// TIA Portal V19 export
FUNCTION_BLOCK "FinalCut_FB"   // FB111, LAD
TITLE = GENERIC OLEODINAMIC HEAD MANAGER
// stored: MemoryReserve 100, SetENOAutomatically false
   VAR_INPUT
      AreaInterface : "AreaInterface";
      ZSI : "udt_ZoneSafetyInterface";
      DSI : "udt_DeviceSafetyInterface";
      DataIn : Struct
         CutHead : "ValveMachine_DataIn";
         DrawHead : "ValveMachine_DataIn";
         MarkHead : "ValveMachine_DataIn";
         Locking : "ValveMachine_DataIn";
         Locking_PressureAI : Int;
      END_STRUCT;
      CIn : Struct
         PressureRunning : Bool := FALSE;
         MaterialStandstill : Bool := FALSE;   // FALSE = Either the movement has already started or is about to start
         EnableCutHead : Bool;
         EnableDrawHead : Bool;
         EnableMarkHead : Bool;
         PPrf_PrgNo : DInt;
         CutHead_Manager : "ValveMachine_Manager";
         DrawHead_Manager : "ValveMachine_Manager";
         MarkHead_Manager : "ValveMachine_Manager";
      END_STRUCT;
      Config : Struct
         CheckRestPosition : Bool := TRUE;
         CutHead : "ValveMachine_Config";
         DrawHead : "ValveMachine_Config";
         MarkHead : "ValveMachine_Config";
         Locking : "ValveMachine_Config";
         Locking_AI_HighLimit : Real;
         Locking_AI_LowLimit : Real;
      END_STRUCT;
   END_VAR
   VAR_OUTPUT
      MachineInterface : "MachineInterface";
      DataOut : Struct
         CutHead : "ValveMachine_DataOut";
         DrawHead : "ValveMachine_DataOut";
         MarkHead : "ValveMachine_DataOut";
         Locking : "ValveMachine_DataOut";
      END_STRUCT;
      COut : Struct
         CutHead : "ValveMachine_COut";
         DrawHead : "ValveMachine_COut";
         MarkHead : "ValveMachine_COut";
         Locking : "ValveMachine_COut";
         Avg_R_to_W_Time : Time;
         Avg_W_to_R_Time : Time;
         AllAtRest : Bool;
      END_STRUCT;
   END_VAR
   VAR_IN_OUT
      PersistentValues : "udt_FinalCut_Pers";
   END_VAR
   VAR
      Sts : Struct
         CycleTime : Struct
            CutHead : Struct
               DT_W_Start : DTL;
               DT_W_Stop : DTL;
               DT_R_Start : DTL;
               DT_R_Stop : DTL;
               R_To_W_Exe : Bool;
               W_To_R_Exe : Bool;
               R_To_W_Items : Int;
               R_To_W_Sum : Time;
               W_To_R_Items : Int;
               W_To_R_Sum : Time;
            END_STRUCT;
            DrawHead : Struct
               DT_W_Start : DTL;
               DT_W_Stop : DTL;
               DT_R_Start : DTL;
               DT_R_Stop : DTL;
               R_To_W_Exe : Bool;
               W_To_R_Exe : Bool;
               R_To_W_Items : Int;
               R_To_W_Sum : Time;
               W_To_R_Items : Int;
               W_To_R_Sum : Time;
            END_STRUCT;
            MarkHead : Struct
               DT_W_Start : DTL;
               DT_W_Stop : DTL;
               DT_R_Start : DTL;
               DT_R_Stop : DTL;
               R_To_W_Exe : Bool;
               W_To_R_Exe : Bool;
               R_To_W_Items : Int;
               R_To_W_Sum : Time;
               W_To_R_Items : Int;
               W_To_R_Sum : Time;
            END_STRUCT;
            PPrf_PrgNoSave : DInt;
         END_STRUCT;
         LockingPressure : Real;
         WorkPressureOk : Bool;
         MinPressureOk : Bool;
      END_STRUCT;
      Ctrl : Struct
         Reload : Struct
            CutHead : Bool;
            DrawHead : Bool;
            MarkHead : Bool;
            Locking : Bool;
         END_STRUCT;
         RstAlarms : Bool;
      END_STRUCT;
      Alarm : Struct
         CutHead : "ValveAlr";
         DrawHead : "ValveAlr";
         MarkHead : "ValveAlr";
         Locking : "ValveAlr";
         Locking_NotAWork : Bool;
      END_STRUCT;
      Warning : Struct
         CutHead : "ValveMachine_Wng";
         DrawHead : "ValveMachine_Wng";
         MarkHead : "ValveMachine_Wng";
         Locking : "ValveMachine_Wng";
         CutHead_NotAtRest : Bool := FALSE;
         DrawHead_NotAtRest : Bool;
         MarkHead_NotAtRest : Bool;
         Locking_NotAWork : Bool;
         MaterialNotStandstill : Bool := FALSE;
      END_STRUCT;
      HMI : Struct
         CutHead : Struct
            Last_R_to_W_ID : DInt;
            Last_R_to_W_Time : Time;
            Last_W_to_R_ID : DInt;
            Last_W_to_R_Time : Time;
            Avg_R_to_W_Time : Time;
            Avg_W_to_R_Time : Time;
            Buffer_R_to_W_Time : Array[1..#BUFFER_ITEMS] of Struct
               ID : DInt;
               Value : Time;
            END_STRUCT;
            Buffer_W_to_R_Time : Array[1..#BUFFER_ITEMS] of Struct
               ID : DInt;
               Value : Time;
            END_STRUCT;
         END_STRUCT;
         DrawHead : Struct
            Last_R_to_W_ID : DInt;
            Last_R_to_W_Time : Time;
            Last_W_to_R_ID : DInt;
            Last_W_to_R_Time : Time;
            Avg_R_to_W_Time : Time;
            Avg_W_to_R_Time : Time;
            Buffer_R_to_W_Time : Array[1..#BUFFER_ITEMS] of Struct
               ID : DInt;
               Value : Time;
            END_STRUCT;
            Buffer_W_to_R_Time : Array[1..#BUFFER_ITEMS] of Struct
               ID : DInt;
               Value : Time;
            END_STRUCT;
         END_STRUCT;
         MarkHead : Struct
            Last_R_to_W_ID : DInt;
            Last_R_to_W_Time : Time;
            Last_W_to_R_ID : DInt;
            Last_W_to_R_Time : Time;
            Avg_R_to_W_Time : Time;
            Avg_W_to_R_Time : Time;
            Buffer_R_to_W_Time : Array[1..#BUFFER_ITEMS] of Struct
               ID : DInt;
               Value : Time;
            END_STRUCT;
            Buffer_W_to_R_Time : Array[1..#BUFFER_ITEMS] of Struct
               ID : DInt;
               Value : Time;
            END_STRUCT;
         END_STRUCT;
      END_STRUCT;
      CutHead : "ValveMachine_FB";
      DrawHead : "ValveMachine_FB";
      MarkHead : "ValveMachine_FB";
      Locking : "ValveMachine_FB";
      TON_CutHead_Pause : IEC_TIMER;
      TON_CutHead_Duration : IEC_TIMER;
      TON_DrawHead_Pause : IEC_TIMER;
      TON_DrawHead_Duration : IEC_TIMER;
      TON_MarkHead_Pause : IEC_TIMER;
      TON_MarkHead_Duration : IEC_TIMER;
      TON_LockingTimeOut : IEC_TIMER;
      PE_Aux : Struct
         CutHead : Struct
            AtRest : Bool;
            AtWork : Bool;
            NotAtRest : Bool;
            NotAtWork : Bool;
         END_STRUCT;
         DrawHead : Struct
            AtRest : Bool;
            AtWork : Bool;
            NotAtRest : Bool;
            NotAtWork : Bool;
         END_STRUCT;
         MarkHead : Struct
            AtRest : Bool;
            AtWork : Bool;
            NotAtRest : Bool;
            NotAtWork : Bool;
         END_STRUCT;
      END_STRUCT;
      i : Int;
   END_VAR
   VAR_TEMP
      PE : Struct
         CutHead : Struct
            AtRest : Bool;
            AtWork : Bool;
            NotAtRest : Bool;
            NotAtWork : Bool;
         END_STRUCT;
         DrawHead : Struct
            AtRest : Bool;
            AtWork : Bool;
            NotAtRest : Bool;
            NotAtWork : Bool;
         END_STRUCT;
         MarkHead : Struct
            AtRest : Bool;
            AtWork : Bool;
            NotAtRest : Bool;
            NotAtWork : Bool;
         END_STRUCT;
      END_STRUCT;
      ReturnVal : Word;
      ScaleRetVal : Word;
   END_VAR
   VAR CONSTANT
      BUFFER_ITEMS : Int := 10;
   END_VAR
   VAR_TEMP   // added for the SCL form of the ladder/FBD networks
      _w1 : Bool;
      _w2 : Bool;
      _w3 : Bool;
      _w4 : Bool;
   END_VAR
BEGIN

REGION Network 1 (SCL): Reset alarms
   #Ctrl.RstAlarms := #AreaInterface.RstAlarms;

   IF    #Ctrl.RstAlarms THEN

       #Alarm.Locking_NotAWork := FALSE;

   END_IF;
END_REGION

REGION Network 2: >
END_REGION

REGION Network 3: <<< CUT HEAD >>>
END_REGION

REGION Network 4: Pressure reload for avoiding losing of rest position cause leakage on hydraulic cylinders
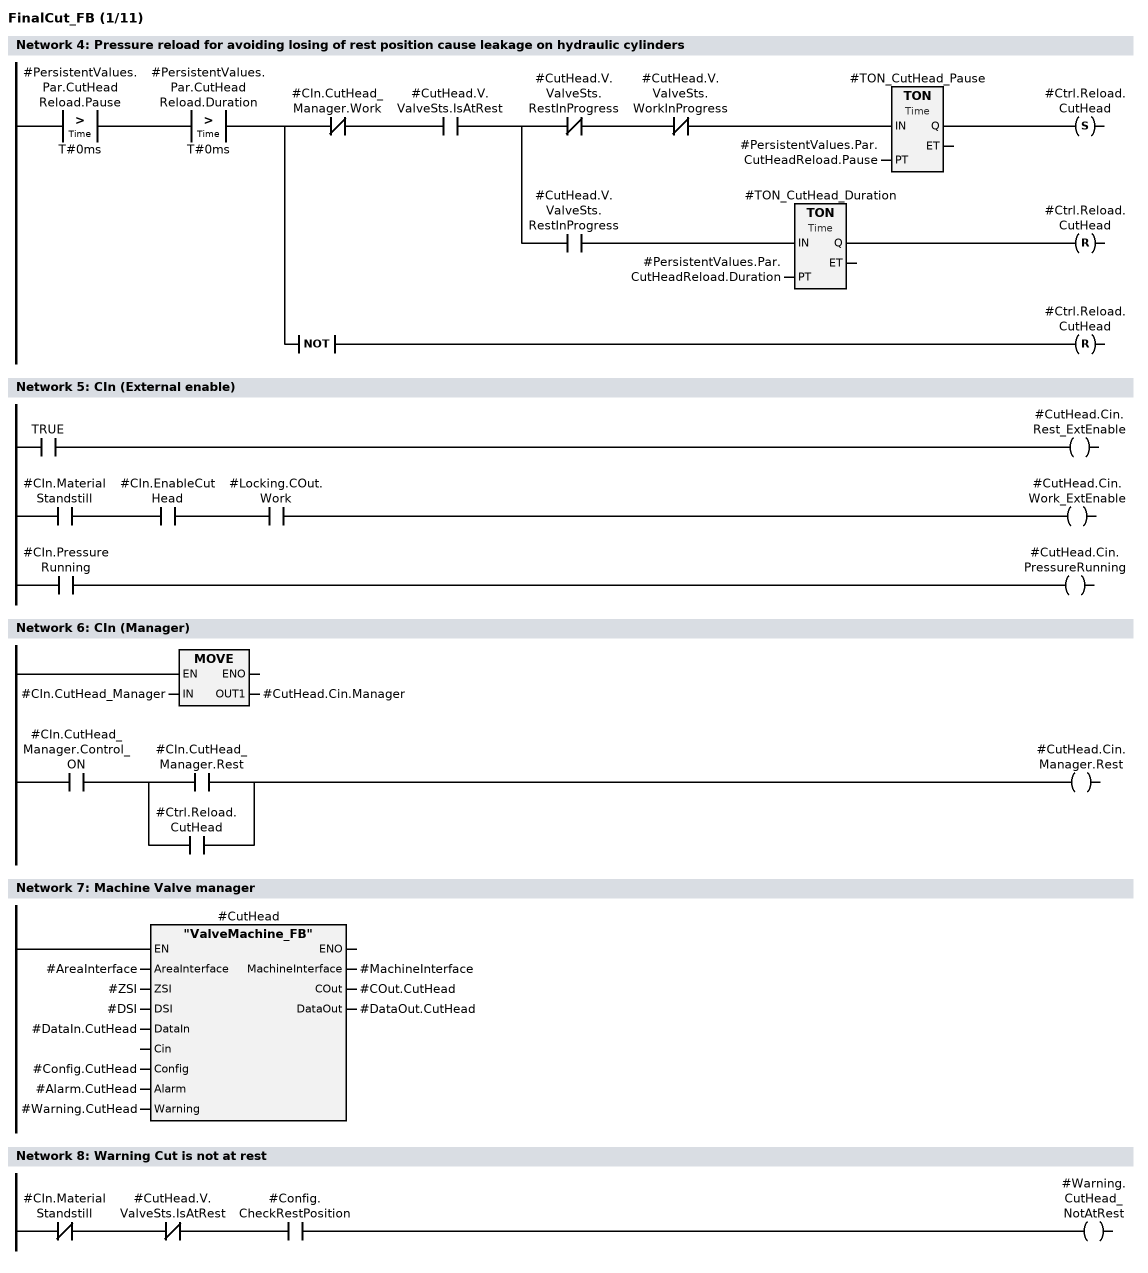
   RUNG wire#powerrail
      { S7_Templates := "SrcType := Time" } GT_Contact(in1 := #PersistentValues.Par.CutHeadReload.Pause, in2 := T#0ms)
      { S7_Templates := "SrcType := Time" } GT_Contact(in1 := #PersistentValues.Par.CutHeadReload.Duration, in2 := T#0ms)
      wire#w1
      I_Contact( #CIn.CutHead_Manager.Work )
      Contact( #CutHead.V.ValveSts.IsAtRest )
      wire#w2
      I_Contact( #CutHead.V.ValveSts.RestInProgress )
      I_Contact( #CutHead.V.ValveSts.WorkInProgress )
      { S7_Templates := "time_type := Time" } #TON_CutHead_Pause.TON(pt := #PersistentValues.Par.CutHeadReload.Pause, et =>)
      S_Coil( #Ctrl.Reload.CutHead )
   END_RUNG
   RUNG wire#w2
      Contact( #CutHead.V.ValveSts.RestInProgress )
      { S7_Templates := "time_type := Time" } #TON_CutHead_Duration.TON(pt := #PersistentValues.Par.CutHeadReload.Duration, et =>)
      R_Coil( #Ctrl.Reload.CutHead )
   END_RUNG
   RUNG wire#w1
      Not()
      R_Coil( #Ctrl.Reload.CutHead )
   END_RUNG
   // the same network as SCL:
   #_w1 := (#PersistentValues.Par.CutHeadReload.Pause > T#0ms) AND (#PersistentValues.Par.CutHeadReload.Duration > T#0ms);
   #_w2 := #_w1 AND NOT #CIn.CutHead_Manager.Work AND #CutHead.V.ValveSts.IsAtRest;
   #TON_CutHead_Pause.TON(IN := #_w2 AND NOT #CutHead.V.ValveSts.RestInProgress AND NOT #CutHead.V.ValveSts.WorkInProgress,
                          PT := #PersistentValues.Par.CutHeadReload.Pause);
   IF #TON_CutHead_Pause.Q THEN #Ctrl.Reload.CutHead := TRUE; END_IF;
   #TON_CutHead_Duration.TON(IN := #_w2 AND #CutHead.V.ValveSts.RestInProgress,
                           PT := #PersistentValues.Par.CutHeadReload.Duration);
   IF #TON_CutHead_Duration.Q THEN #Ctrl.Reload.CutHead := FALSE; END_IF;
   IF NOT #_w1 THEN #Ctrl.Reload.CutHead := FALSE; END_IF;
END_REGION

REGION Network 5: CIn (External enable)
   RUNG wire#powerrail
      Contact( TRUE )
      Coil( #CutHead.Cin.Rest_ExtEnable )
   END_RUNG
   RUNG wire#powerrail
      Contact( #CIn.MaterialStandstill )
      Contact( #CIn.EnableCutHead )
      Contact( #Locking.COut.Work )
      Coil( #CutHead.Cin.Work_ExtEnable )
   END_RUNG
   RUNG wire#powerrail
      Contact( #CIn.PressureRunning )
      Coil( #CutHead.Cin.PressureRunning )
   END_RUNG
   // the same network as SCL:
   #CutHead.Cin.Rest_ExtEnable := TRUE;
   #CutHead.Cin.Work_ExtEnable := #CIn.MaterialStandstill AND #CIn.EnableCutHead AND #Locking.COut.Work;
   #CutHead.Cin.PressureRunning := #CIn.PressureRunning;
END_REGION

REGION Network 6: CIn (Manager)
   RUNG wire#powerrail
      Move(in := #CIn.CutHead_Manager, out1 => #CutHead.Cin.Manager)
   END_RUNG
   RUNG wire#powerrail
      Contact( #CIn.CutHead_Manager.Control_ON )
      wire#w1
      Contact( #CIn.CutHead_Manager.Rest )
      wire#w2
      Coil( #CutHead.Cin.Manager.Rest )
   END_RUNG
   RUNG wire#w1
      Contact( #Ctrl.Reload.CutHead )
   END_RUNG wire#w2
   // the same network as SCL:
   #CutHead.Cin.Manager := #CIn.CutHead_Manager;
   #CutHead.Cin.Manager.Rest := #CIn.CutHead_Manager.Control_ON AND (#CIn.CutHead_Manager.Rest OR #Ctrl.Reload.CutHead);
END_REGION

REGION Network 7: Machine Valve manager
   RUNG wire#powerrail
      #CutHead(AreaInterface := #AreaInterface, ZSI := #ZSI, DSI := #DSI, DataIn := #DataIn.CutHead, Cin :=, Config := #Config.CutHead, Alarm := #Alarm.CutHead, Warning := #Warning.CutHead, MachineInterface => #MachineInterface, COut => #COut.CutHead, DataOut => #DataOut.CutHead)
   END_RUNG
   // the same network as SCL:
   #CutHead(AreaInterface := #AreaInterface,   // "ValveMachine_FB"
            ZSI := #ZSI,
            DSI := #DSI,
            DataIn := #DataIn.CutHead,
            Config := #Config.CutHead,
            Alarm := #Alarm.CutHead,
            Warning := #Warning.CutHead,
            MachineInterface => #MachineInterface,
            COut => #COut.CutHead,
            DataOut => #DataOut.CutHead);
END_REGION

REGION Network 8: Warning Cut is not at rest
   RUNG wire#powerrail
      I_Contact( #CIn.MaterialStandstill )
      I_Contact( #CutHead.V.ValveSts.IsAtRest )
      Contact( #Config.CheckRestPosition )
      Coil( #Warning.CutHead_NotAtRest )
   END_RUNG
   // the same network as SCL:
   #Warning.CutHead_NotAtRest := NOT #CIn.MaterialStandstill AND NOT #CutHead.V.ValveSts.IsAtRest AND #Config.CheckRestPosition;
END_REGION

REGION Network 9: At Rest / At work positive/negative edge
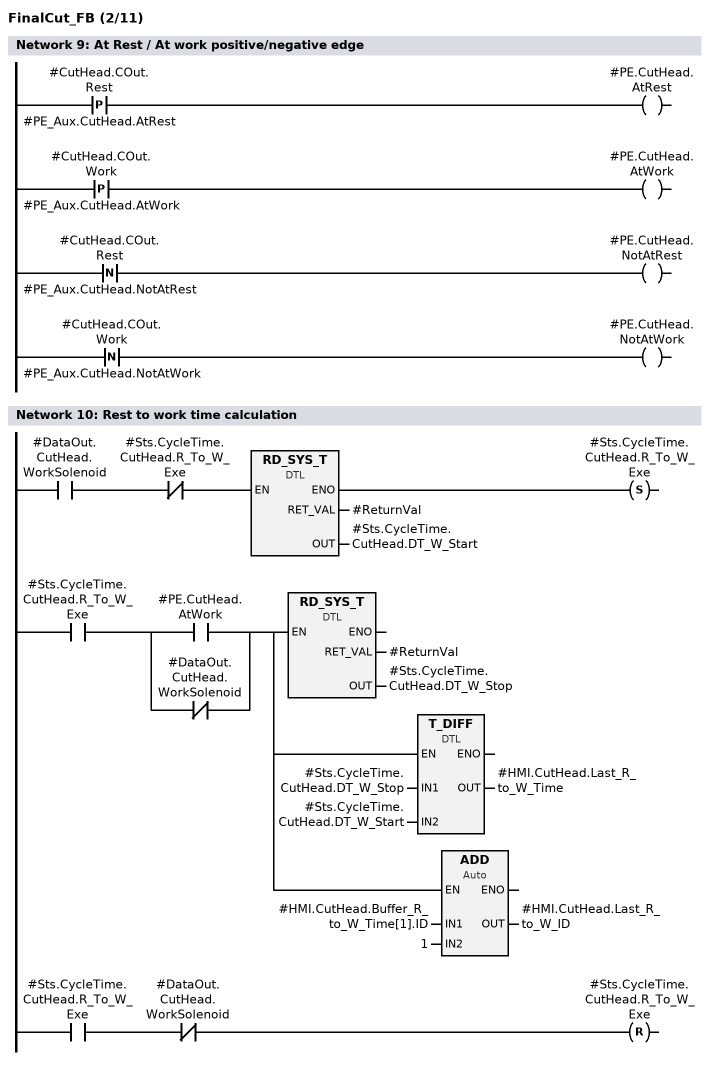
   RUNG wire#powerrail
      P_Contact(operand := #CutHead.COut.Rest, bit := #PE_Aux.CutHead.AtRest)
      Coil( #PE.CutHead.AtRest )
   END_RUNG
   RUNG wire#powerrail
      P_Contact(operand := #CutHead.COut.Work, bit := #PE_Aux.CutHead.AtWork)
      Coil( #PE.CutHead.AtWork )
   END_RUNG
   RUNG wire#powerrail
      N_Contact(operand := #CutHead.COut.Rest, bit := #PE_Aux.CutHead.NotAtRest)
      Coil( #PE.CutHead.NotAtRest )
   END_RUNG
   RUNG wire#powerrail
      N_Contact(operand := #CutHead.COut.Work, bit := #PE_Aux.CutHead.NotAtWork)
      Coil( #PE.CutHead.NotAtWork )
   END_RUNG
   // the same network as SCL:
   #_w1 := #CutHead.COut.Rest AND NOT #PE_Aux.CutHead.AtRest;   // rising edge of #CutHead.COut.Rest
   #PE_Aux.CutHead.AtRest := #CutHead.COut.Rest;
   #PE.CutHead.AtRest := #_w1;
   #_w2 := #CutHead.COut.Work AND NOT #PE_Aux.CutHead.AtWork;   // rising edge of #CutHead.COut.Work
   #PE_Aux.CutHead.AtWork := #CutHead.COut.Work;
   #PE.CutHead.AtWork := #_w2;
   #_w3 := NOT #CutHead.COut.Rest AND #PE_Aux.CutHead.NotAtRest;   // falling edge of #CutHead.COut.Rest
   #PE_Aux.CutHead.NotAtRest := #CutHead.COut.Rest;
   #PE.CutHead.NotAtRest := #_w3;
   #_w4 := NOT #CutHead.COut.Work AND #PE_Aux.CutHead.NotAtWork;   // falling edge of #CutHead.COut.Work
   #PE_Aux.CutHead.NotAtWork := #CutHead.COut.Work;
   #PE.CutHead.NotAtWork := #_w4;
END_REGION

REGION Network 10: Rest to work time calculation
   RUNG wire#powerrail
      Contact( #DataOut.CutHead.WorkSolenoid )
      I_Contact( #Sts.CycleTime.CutHead.R_To_W_Exe )
      { S7_Templates := "date_type := DTL" } RD_SYS_T(RET_VAL => #ReturnVal, OUT => #Sts.CycleTime.CutHead.DT_W_Start)
      S_Coil( #Sts.CycleTime.CutHead.R_To_W_Exe )
   END_RUNG
   RUNG wire#powerrail
      Contact( #Sts.CycleTime.CutHead.R_To_W_Exe )
      wire#w1
      Contact( #PE.CutHead.AtWork )
      wire#w2
      { S7_Templates := "date_type := DTL" } RD_SYS_T(RET_VAL => #ReturnVal, OUT => #Sts.CycleTime.CutHead.DT_W_Stop)
   END_RUNG
   RUNG wire#w1
      I_Contact( #DataOut.CutHead.WorkSolenoid )
   END_RUNG wire#w2
   RUNG wire#w2
      { S7_Templates := "[date_type := DTL, time_type := Time]" } T_DIFF(IN1 := #Sts.CycleTime.CutHead.DT_W_Stop, IN2 := #Sts.CycleTime.CutHead.DT_W_Start, OUT => #HMI.CutHead.Last_R_to_W_Time)
   END_RUNG
   RUNG wire#w2
      Add(in1 := #HMI.CutHead.Buffer_R_to_W_Time[1].ID, in2 := 1, out => #HMI.CutHead.Last_R_to_W_ID)
   END_RUNG
   RUNG wire#powerrail
      Contact( #Sts.CycleTime.CutHead.R_To_W_Exe )
      I_Contact( #DataOut.CutHead.WorkSolenoid )
      R_Coil( #Sts.CycleTime.CutHead.R_To_W_Exe )
   END_RUNG
   // the same network as SCL:
   #ReturnVal := RD_SYS_T(EN := #DataOut.CutHead.WorkSolenoid AND NOT #Sts.CycleTime.CutHead.R_To_W_Exe,
                          OUT => #Sts.CycleTime.CutHead.DT_W_Start,
                          ENO => #_w1);
   IF #_w1 THEN #Sts.CycleTime.CutHead.R_To_W_Exe := TRUE; END_IF;
   IF #Sts.CycleTime.CutHead.R_To_W_Exe AND (#PE.CutHead.AtWork OR NOT #DataOut.CutHead.WorkSolenoid) THEN
       #ReturnVal := RD_SYS_T(OUT => #Sts.CycleTime.CutHead.DT_W_Stop);
       T_DIFF(IN1 := #Sts.CycleTime.CutHead.DT_W_Stop,
              IN2 := #Sts.CycleTime.CutHead.DT_W_Start,
              OUT => #HMI.CutHead.Last_R_to_W_Time);
       #HMI.CutHead.Last_R_to_W_ID := #HMI.CutHead.Buffer_R_to_W_Time[1].ID + 1;
   END_IF;
   IF #Sts.CycleTime.CutHead.R_To_W_Exe AND NOT #DataOut.CutHead.WorkSolenoid THEN
       #Sts.CycleTime.CutHead.R_To_W_Exe := FALSE;
   END_IF;
END_REGION

REGION Network 11: Work to rest time calculation
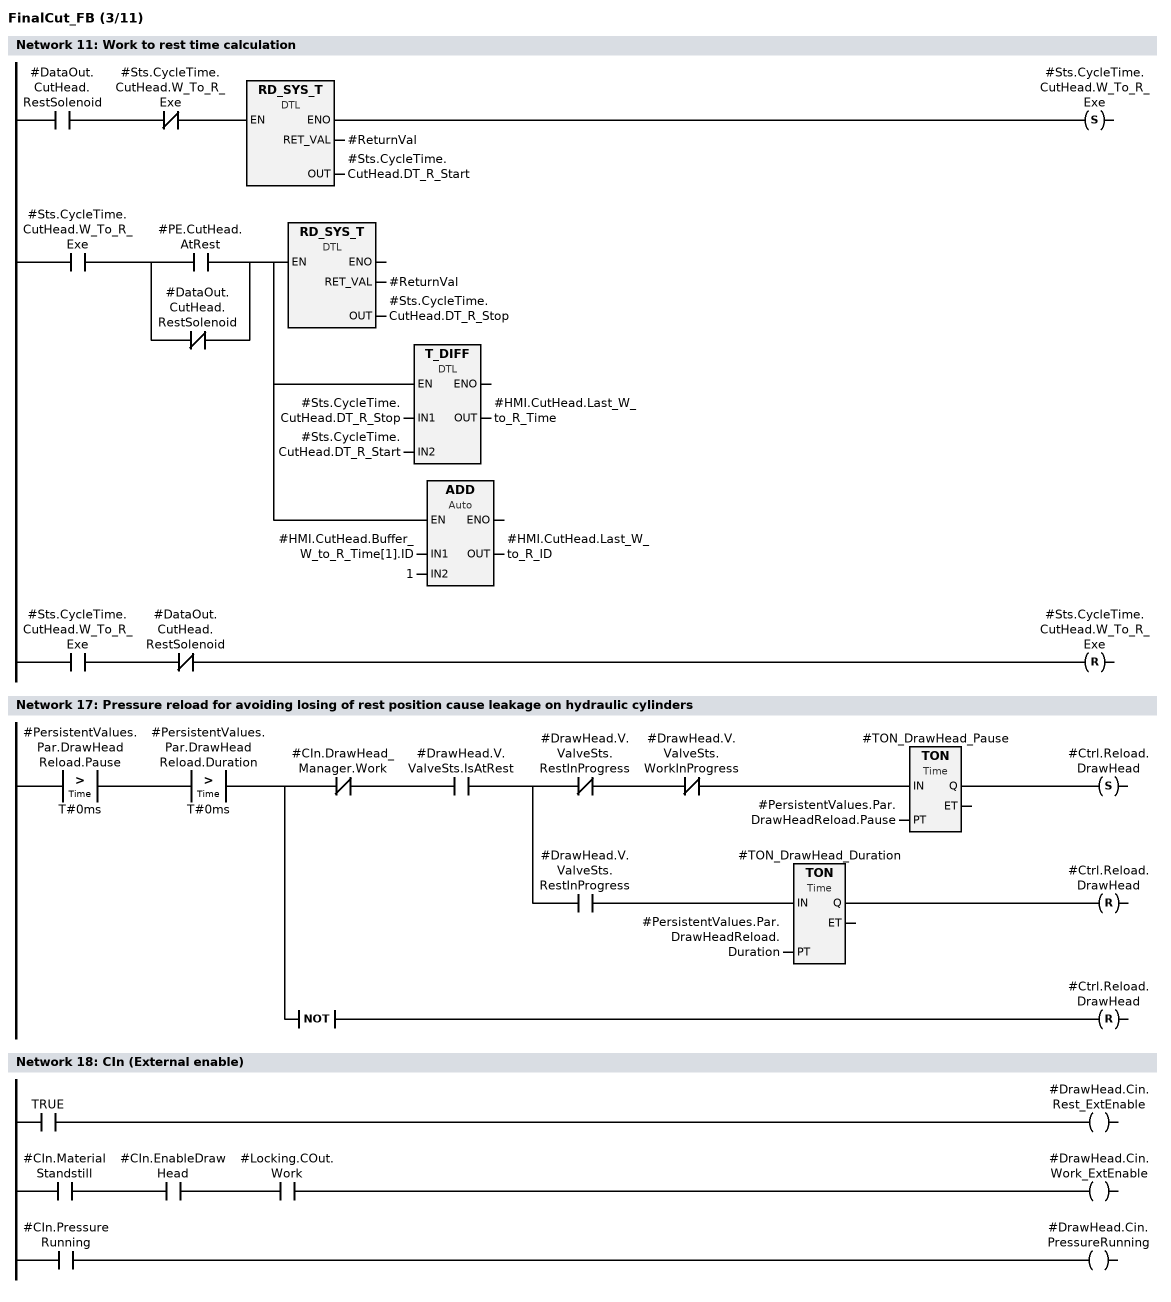
   RUNG wire#powerrail
      Contact( #DataOut.CutHead.RestSolenoid )
      I_Contact( #Sts.CycleTime.CutHead.W_To_R_Exe )
      { S7_Templates := "date_type := DTL" } RD_SYS_T(RET_VAL => #ReturnVal, OUT => #Sts.CycleTime.CutHead.DT_R_Start)
      S_Coil( #Sts.CycleTime.CutHead.W_To_R_Exe )
   END_RUNG
   RUNG wire#powerrail
      Contact( #Sts.CycleTime.CutHead.W_To_R_Exe )
      wire#w1
      Contact( #PE.CutHead.AtRest )
      wire#w2
      { S7_Templates := "date_type := DTL" } RD_SYS_T(RET_VAL => #ReturnVal, OUT => #Sts.CycleTime.CutHead.DT_R_Stop)
   END_RUNG
   RUNG wire#w1
      I_Contact( #DataOut.CutHead.RestSolenoid )
   END_RUNG wire#w2
   RUNG wire#w2
      { S7_Templates := "[date_type := DTL, time_type := Time]" } T_DIFF(IN1 := #Sts.CycleTime.CutHead.DT_R_Stop, IN2 := #Sts.CycleTime.CutHead.DT_R_Start, OUT => #HMI.CutHead.Last_W_to_R_Time)
   END_RUNG
   RUNG wire#w2
      Add(in1 := #HMI.CutHead.Buffer_W_to_R_Time[1].ID, in2 := 1, out => #HMI.CutHead.Last_W_to_R_ID)
   END_RUNG
   RUNG wire#powerrail
      Contact( #Sts.CycleTime.CutHead.W_To_R_Exe )
      I_Contact( #DataOut.CutHead.RestSolenoid )
      R_Coil( #Sts.CycleTime.CutHead.W_To_R_Exe )
   END_RUNG
   // the same network as SCL:
   #ReturnVal := RD_SYS_T(EN := #DataOut.CutHead.RestSolenoid AND NOT #Sts.CycleTime.CutHead.W_To_R_Exe,
                          OUT => #Sts.CycleTime.CutHead.DT_R_Start,
                          ENO => #_w1);
   IF #_w1 THEN #Sts.CycleTime.CutHead.W_To_R_Exe := TRUE; END_IF;
   IF #Sts.CycleTime.CutHead.W_To_R_Exe AND (#PE.CutHead.AtRest OR NOT #DataOut.CutHead.RestSolenoid) THEN
       #ReturnVal := RD_SYS_T(OUT => #Sts.CycleTime.CutHead.DT_R_Stop);
       T_DIFF(IN1 := #Sts.CycleTime.CutHead.DT_R_Stop,
              IN2 := #Sts.CycleTime.CutHead.DT_R_Start,
              OUT => #HMI.CutHead.Last_W_to_R_Time);
       #HMI.CutHead.Last_W_to_R_ID := #HMI.CutHead.Buffer_W_to_R_Time[1].ID + 1;
   END_IF;
   IF #Sts.CycleTime.CutHead.W_To_R_Exe AND NOT #DataOut.CutHead.RestSolenoid THEN
       #Sts.CycleTime.CutHead.W_To_R_Exe := FALSE;
   END_IF;
END_REGION

REGION Network 12 (SCL): Init buffers & average calculations
   IF #CIn.PPrf_PrgNo <> #Sts.CycleTime.PPrf_PrgNoSave OR #CIn.PPrf_PrgNo <= 0 THEN

       FOR #i := 1 TO #BUFFER_ITEMS DO
           #HMI.CutHead.Buffer_R_to_W_Time[#i].ID := 0;
           #HMI.CutHead.Buffer_R_to_W_Time[#i].Value := T#0s;
           #HMI.CutHead.Buffer_W_to_R_Time[#i].ID := 0;
           #HMI.CutHead.Buffer_W_to_R_Time[#i].Value := T#0s;
       END_FOR;

       #HMI.CutHead.Last_R_to_W_ID := 0;
       #HMI.CutHead.Last_R_to_W_Time := T#0ms;
       #HMI.CutHead.Avg_R_to_W_Time := #Config.CutHead.V.WorkTimeOut;

       #HMI.CutHead.Last_W_to_R_ID := 0;
       #HMI.CutHead.Last_W_to_R_Time := T#0ms;
       #HMI.CutHead.Avg_W_to_R_Time := #Config.CutHead.V.RestTimeOut;

   END_IF;


   #Sts.CycleTime.PPrf_PrgNoSave := #CIn.PPrf_PrgNo;
END_REGION

REGION Network 13 (SCL): Add new items to Rest-TO-Work buffer & calculate average

   IF #HMI.CutHead.Last_R_to_W_Time >= #CutHead.Config.V.WorkTimeOut OR #Alarm.CutHead.TimeOutWork THEN

       #HMI.CutHead.Last_R_to_W_ID := -1; // Force red background on the HMI visualization



   ELSIF #HMI.CutHead.Last_R_to_W_ID <> #HMI.CutHead.Buffer_R_to_W_Time[1].ID AND #HMI.CutHead.Last_R_to_W_Time < #CutHead.Config.V.WorkTimeOut AND #HMI.CutHead.Last_R_to_W_Time > T#0ms THEN

       #i := #BUFFER_ITEMS;

       WHILE #i >= 2 DO

           #HMI.CutHead.Buffer_R_to_W_Time[#i] := #HMI.CutHead.Buffer_R_to_W_Time[#i - 1];

           #i -= 1;

       END_WHILE;

       #HMI.CutHead.Buffer_R_to_W_Time[1].ID := #HMI.CutHead.Last_R_to_W_ID;
       #HMI.CutHead.Buffer_R_to_W_Time[1].Value := #HMI.CutHead.Last_R_to_W_Time;

       #Sts.CycleTime.CutHead.R_To_W_Items := 0;
       #Sts.CycleTime.CutHead.R_To_W_Sum := T#0s;


       FOR #i := 1 TO #BUFFER_ITEMS DO

           IF #HMI.CutHead.Buffer_R_to_W_Time[#i].ID > 0 AND #HMI.CutHead.Buffer_R_to_W_Time[#i].Value > T#0ms THEN
               #Sts.CycleTime.CutHead.R_To_W_Items += 1;
               #Sts.CycleTime.CutHead.R_To_W_Sum := #Sts.CycleTime.CutHead.R_To_W_Sum + #HMI.CutHead.Buffer_R_to_W_Time[#i].Value;
           END_IF;

       END_FOR;

       IF #Sts.CycleTime.CutHead.R_To_W_Items >= 5 THEN
           #HMI.CutHead.Avg_R_to_W_Time := #Sts.CycleTime.CutHead.R_To_W_Sum / #Sts.CycleTime.CutHead.R_To_W_Items;
       ELSE
           #HMI.CutHead.Avg_R_to_W_Time := #Config.CutHead.V.WorkTimeOut;
       END_IF;

   END_IF;
END_REGION

REGION Network 14 (SCL): Add new items to Work-TO-Rest buffer & calculate average
   IF #HMI.CutHead.Last_W_to_R_Time >= #CutHead.Config.V.RestTimeOut OR #Alarm.CutHead.TimeOutRest THEN

       #HMI.CutHead.Last_W_to_R_ID := -1; // Force red background on the HMI visualization

   ELSIF #HMI.CutHead.Last_W_to_R_ID <> #HMI.CutHead.Buffer_W_to_R_Time[1].ID AND #HMI.CutHead.Last_W_to_R_Time < #CutHead.Config.V.RestTimeOut AND #HMI.CutHead.Last_W_to_R_Time > T#0ms  THEN

       #i := #BUFFER_ITEMS;

       WHILE #i >= 2 DO

           #HMI.CutHead.Buffer_W_to_R_Time[#i] := #HMI.CutHead.Buffer_W_to_R_Time[#i - 1];

           #i -= 1;

       END_WHILE;

       #HMI.CutHead.Buffer_W_to_R_Time[1].ID := #HMI.CutHead.Last_W_to_R_ID;
       #HMI.CutHead.Buffer_W_to_R_Time[1].Value := #HMI.CutHead.Last_W_to_R_Time;

       #Sts.CycleTime.CutHead.W_To_R_Items := 0;
       #Sts.CycleTime.CutHead.W_To_R_Sum := T#0s;


       FOR #i := 1 TO #BUFFER_ITEMS DO

           IF #HMI.CutHead.Buffer_W_to_R_Time[#i].ID > 0 AND #HMI.CutHead.Buffer_W_to_R_Time[#i].Value > T#0ms  THEN
               #Sts.CycleTime.CutHead.W_To_R_Items += 1;
               #Sts.CycleTime.CutHead.W_To_R_Sum := #Sts.CycleTime.CutHead.W_To_R_Sum + #HMI.CutHead.Buffer_W_to_R_Time[#i].Value;
           END_IF;

       END_FOR;

       IF #Sts.CycleTime.CutHead.W_To_R_Items >= 5 THEN
           #HMI.CutHead.Avg_W_to_R_Time := #Sts.CycleTime.CutHead.W_To_R_Sum / #Sts.CycleTime.CutHead.W_To_R_Items;
       ELSE
           #HMI.CutHead.Avg_W_to_R_Time := #Config.CutHead.V.RestTimeOut;
       END_IF;

   END_IF;
END_REGION

REGION Network 15: >
END_REGION

REGION Network 16: <<< DRAWING HEAD >>>
END_REGION

REGION Network 17: Pressure reload for avoiding losing of rest position cause leakage on hydraulic cylinders
   RUNG wire#powerrail
      { S7_Templates := "SrcType := Time" } GT_Contact(in1 := #PersistentValues.Par.DrawHeadReload.Pause, in2 := T#0ms)
      { S7_Templates := "SrcType := Time" } GT_Contact(in1 := #PersistentValues.Par.DrawHeadReload.Duration, in2 := T#0ms)
      wire#w1
      I_Contact( #CIn.DrawHead_Manager.Work )
      Contact( #DrawHead.V.ValveSts.IsAtRest )
      wire#w2
      I_Contact( #DrawHead.V.ValveSts.RestInProgress )
      I_Contact( #DrawHead.V.ValveSts.WorkInProgress )
      { S7_Templates := "time_type := Time" } #TON_DrawHead_Pause.TON(pt := #PersistentValues.Par.DrawHeadReload.Pause, et =>)
      S_Coil( #Ctrl.Reload.DrawHead )
   END_RUNG
   RUNG wire#w2
      Contact( #DrawHead.V.ValveSts.RestInProgress )
      { S7_Templates := "time_type := Time" } #TON_DrawHead_Duration.TON(pt := #PersistentValues.Par.DrawHeadReload.Duration, et =>)
      R_Coil( #Ctrl.Reload.DrawHead )
   END_RUNG
   RUNG wire#w1
      Not()
      R_Coil( #Ctrl.Reload.DrawHead )
   END_RUNG
   // the same network as SCL:
   #_w1 := (#PersistentValues.Par.DrawHeadReload.Pause > T#0ms) AND (#PersistentValues.Par.DrawHeadReload.Duration > T#0ms);
   #_w2 := #_w1 AND NOT #CIn.DrawHead_Manager.Work AND #DrawHead.V.ValveSts.IsAtRest;
   #TON_DrawHead_Pause.TON(IN := #_w2 AND NOT #DrawHead.V.ValveSts.RestInProgress AND NOT #DrawHead.V.ValveSts.WorkInProgress,
                           PT := #PersistentValues.Par.DrawHeadReload.Pause);
   IF #TON_DrawHead_Pause.Q THEN #Ctrl.Reload.DrawHead := TRUE; END_IF;
   #TON_DrawHead_Duration.TON(IN := #_w2 AND #DrawHead.V.ValveSts.RestInProgress,
                           PT := #PersistentValues.Par.DrawHeadReload.Duration);
   IF #TON_DrawHead_Duration.Q THEN #Ctrl.Reload.DrawHead := FALSE; END_IF;
   IF NOT #_w1 THEN #Ctrl.Reload.DrawHead := FALSE; END_IF;
END_REGION

REGION Network 18: CIn (External enable)
   RUNG wire#powerrail
      Contact( TRUE )
      Coil( #DrawHead.Cin.Rest_ExtEnable )
   END_RUNG
   RUNG wire#powerrail
      Contact( #CIn.MaterialStandstill )
      Contact( #CIn.EnableDrawHead )
      Contact( #Locking.COut.Work )
      Coil( #DrawHead.Cin.Work_ExtEnable )
   END_RUNG
   RUNG wire#powerrail
      Contact( #CIn.PressureRunning )
      Coil( #DrawHead.Cin.PressureRunning )
   END_RUNG
   // the same network as SCL:
   #DrawHead.Cin.Rest_ExtEnable := TRUE;
   #DrawHead.Cin.Work_ExtEnable := #CIn.MaterialStandstill AND #CIn.EnableDrawHead AND #Locking.COut.Work;
   #DrawHead.Cin.PressureRunning := #CIn.PressureRunning;
END_REGION

REGION Network 19: CIn (Manager)
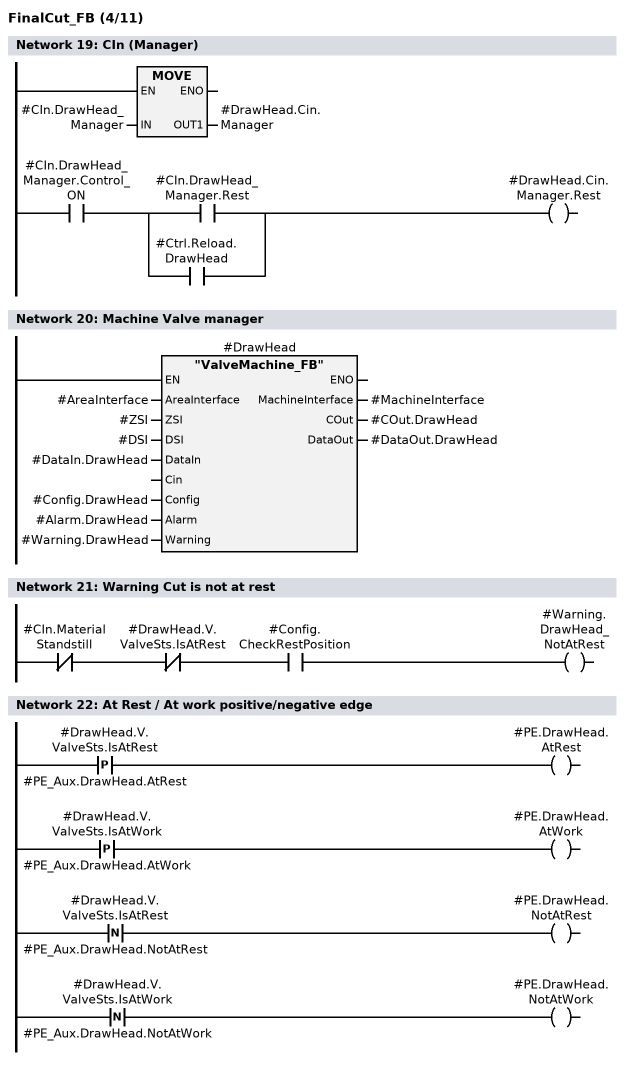
   RUNG wire#powerrail
      Move(in := #CIn.DrawHead_Manager, out1 => #DrawHead.Cin.Manager)
   END_RUNG
   RUNG wire#powerrail
      Contact( #CIn.DrawHead_Manager.Control_ON )
      wire#w1
      Contact( #CIn.DrawHead_Manager.Rest )
      wire#w2
      Coil( #DrawHead.Cin.Manager.Rest )
   END_RUNG
   RUNG wire#w1
      Contact( #Ctrl.Reload.DrawHead )
   END_RUNG wire#w2
   // the same network as SCL:
   #DrawHead.Cin.Manager := #CIn.DrawHead_Manager;
   #DrawHead.Cin.Manager.Rest := #CIn.DrawHead_Manager.Control_ON AND (#CIn.DrawHead_Manager.Rest OR #Ctrl.Reload.DrawHead);
END_REGION

REGION Network 20: Machine Valve manager
   RUNG wire#powerrail
      #DrawHead(AreaInterface := #AreaInterface, ZSI := #ZSI, DSI := #DSI, DataIn := #DataIn.DrawHead, Cin :=, Config := #Config.DrawHead, Alarm := #Alarm.DrawHead, Warning := #Warning.DrawHead, MachineInterface => #MachineInterface, COut => #COut.DrawHead, DataOut => #DataOut.DrawHead)
   END_RUNG
   // the same network as SCL:
   #DrawHead(AreaInterface := #AreaInterface,   // "ValveMachine_FB"
             ZSI := #ZSI,
             DSI := #DSI,
             DataIn := #DataIn.DrawHead,
             Config := #Config.DrawHead,
             Alarm := #Alarm.DrawHead,
             Warning := #Warning.DrawHead,
             MachineInterface => #MachineInterface,
             COut => #COut.DrawHead,
             DataOut => #DataOut.DrawHead);
END_REGION

REGION Network 21: Warning Cut is not at rest
   RUNG wire#powerrail
      I_Contact( #CIn.MaterialStandstill )
      I_Contact( #DrawHead.V.ValveSts.IsAtRest )
      Contact( #Config.CheckRestPosition )
      Coil( #Warning.DrawHead_NotAtRest )
   END_RUNG
   // the same network as SCL:
   #Warning.DrawHead_NotAtRest := NOT #CIn.MaterialStandstill AND NOT #DrawHead.V.ValveSts.IsAtRest AND #Config.CheckRestPosition;
END_REGION

REGION Network 22: At Rest / At work positive/negative edge
   RUNG wire#powerrail
      P_Contact(operand := #DrawHead.V.ValveSts.IsAtRest, bit := #PE_Aux.DrawHead.AtRest)
      Coil( #PE.DrawHead.AtRest )
   END_RUNG
   RUNG wire#powerrail
      P_Contact(operand := #DrawHead.V.ValveSts.IsAtWork, bit := #PE_Aux.DrawHead.AtWork)
      Coil( #PE.DrawHead.AtWork )
   END_RUNG
   RUNG wire#powerrail
      N_Contact(operand := #DrawHead.V.ValveSts.IsAtRest, bit := #PE_Aux.DrawHead.NotAtRest)
      Coil( #PE.DrawHead.NotAtRest )
   END_RUNG
   RUNG wire#powerrail
      N_Contact(operand := #DrawHead.V.ValveSts.IsAtWork, bit := #PE_Aux.DrawHead.NotAtWork)
      Coil( #PE.DrawHead.NotAtWork )
   END_RUNG
   // the same network as SCL:
   #_w1 := #DrawHead.V.ValveSts.IsAtRest AND NOT #PE_Aux.DrawHead.AtRest;   // rising edge of #DrawHead.V.ValveSts.IsAtRest
   #PE_Aux.DrawHead.AtRest := #DrawHead.V.ValveSts.IsAtRest;
   #PE.DrawHead.AtRest := #_w1;
   #_w2 := #DrawHead.V.ValveSts.IsAtWork AND NOT #PE_Aux.DrawHead.AtWork;   // rising edge of #DrawHead.V.ValveSts.IsAtWork
   #PE_Aux.DrawHead.AtWork := #DrawHead.V.ValveSts.IsAtWork;
   #PE.DrawHead.AtWork := #_w2;
   #_w3 := NOT #DrawHead.V.ValveSts.IsAtRest AND #PE_Aux.DrawHead.NotAtRest;   // falling edge of #DrawHead.V.ValveSts.IsAtRest
   #PE_Aux.DrawHead.NotAtRest := #DrawHead.V.ValveSts.IsAtRest;
   #PE.DrawHead.NotAtRest := #_w3;
   #_w4 := NOT #DrawHead.V.ValveSts.IsAtWork AND #PE_Aux.DrawHead.NotAtWork;   // falling edge of #DrawHead.V.ValveSts.IsAtWork
   #PE_Aux.DrawHead.NotAtWork := #DrawHead.V.ValveSts.IsAtWork;
   #PE.DrawHead.NotAtWork := #_w4;
END_REGION

REGION Network 23: Rest to work time calculation
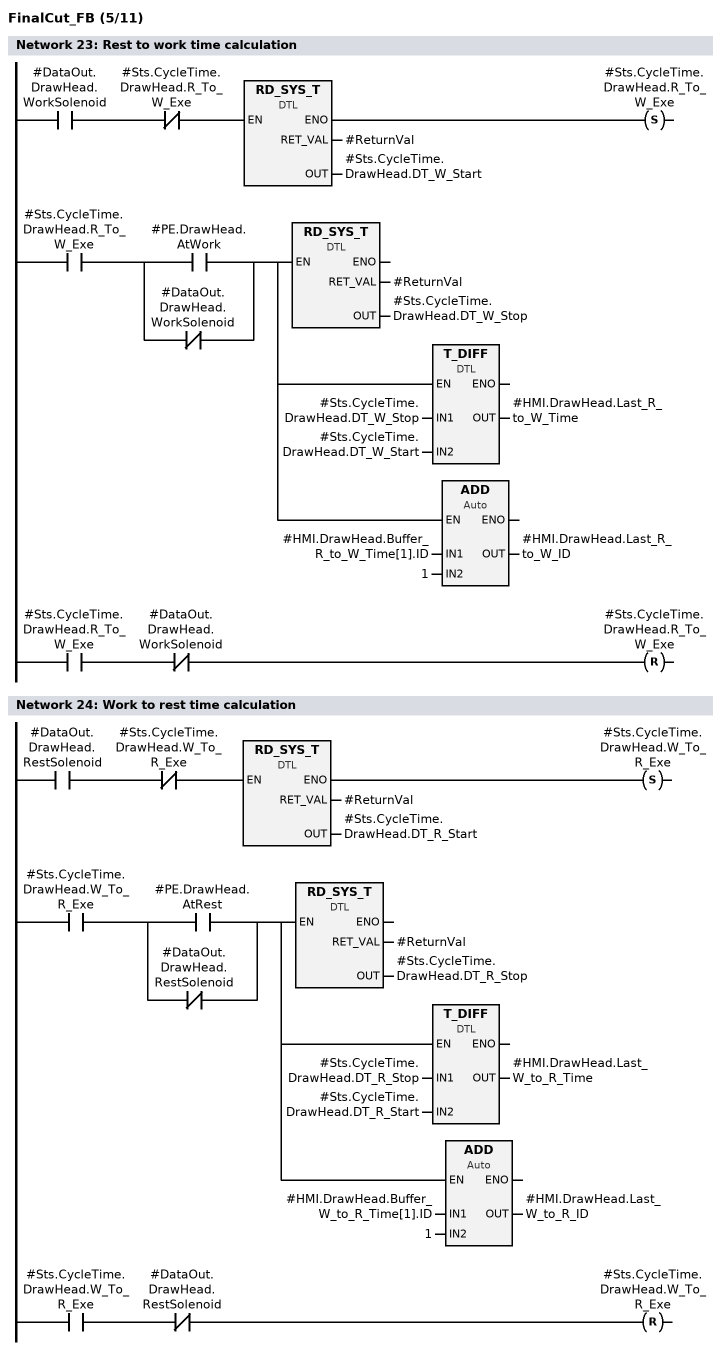
   RUNG wire#powerrail
      Contact( #DataOut.DrawHead.WorkSolenoid )
      I_Contact( #Sts.CycleTime.DrawHead.R_To_W_Exe )
      { S7_Templates := "date_type := DTL" } RD_SYS_T(RET_VAL => #ReturnVal, OUT => #Sts.CycleTime.DrawHead.DT_W_Start)
      S_Coil( #Sts.CycleTime.DrawHead.R_To_W_Exe )
   END_RUNG
   RUNG wire#powerrail
      Contact( #Sts.CycleTime.DrawHead.R_To_W_Exe )
      wire#w1
      Contact( #PE.DrawHead.AtWork )
      wire#w2
      { S7_Templates := "date_type := DTL" } RD_SYS_T(RET_VAL => #ReturnVal, OUT => #Sts.CycleTime.DrawHead.DT_W_Stop)
   END_RUNG
   RUNG wire#w1
      I_Contact( #DataOut.DrawHead.WorkSolenoid )
   END_RUNG wire#w2
   RUNG wire#w2
      { S7_Templates := "[date_type := DTL, time_type := Time]" } T_DIFF(IN1 := #Sts.CycleTime.DrawHead.DT_W_Stop, IN2 := #Sts.CycleTime.DrawHead.DT_W_Start, OUT => #HMI.DrawHead.Last_R_to_W_Time)
   END_RUNG
   RUNG wire#w2
      Add(in1 := #HMI.DrawHead.Buffer_R_to_W_Time[1].ID, in2 := 1, out => #HMI.DrawHead.Last_R_to_W_ID)
   END_RUNG
   RUNG wire#powerrail
      Contact( #Sts.CycleTime.DrawHead.R_To_W_Exe )
      I_Contact( #DataOut.DrawHead.WorkSolenoid )
      R_Coil( #Sts.CycleTime.DrawHead.R_To_W_Exe )
   END_RUNG
   // the same network as SCL:
   #ReturnVal := RD_SYS_T(EN := #DataOut.DrawHead.WorkSolenoid AND NOT #Sts.CycleTime.DrawHead.R_To_W_Exe,
                          OUT => #Sts.CycleTime.DrawHead.DT_W_Start,
                          ENO => #_w1);
   IF #_w1 THEN #Sts.CycleTime.DrawHead.R_To_W_Exe := TRUE; END_IF;
   IF #Sts.CycleTime.DrawHead.R_To_W_Exe AND (#PE.DrawHead.AtWork OR NOT #DataOut.DrawHead.WorkSolenoid) THEN
       #ReturnVal := RD_SYS_T(OUT => #Sts.CycleTime.DrawHead.DT_W_Stop);
       T_DIFF(IN1 := #Sts.CycleTime.DrawHead.DT_W_Stop,
              IN2 := #Sts.CycleTime.DrawHead.DT_W_Start,
              OUT => #HMI.DrawHead.Last_R_to_W_Time);
       #HMI.DrawHead.Last_R_to_W_ID := #HMI.DrawHead.Buffer_R_to_W_Time[1].ID + 1;
   END_IF;
   IF #Sts.CycleTime.DrawHead.R_To_W_Exe AND NOT #DataOut.DrawHead.WorkSolenoid THEN
       #Sts.CycleTime.DrawHead.R_To_W_Exe := FALSE;
   END_IF;
END_REGION

REGION Network 24: Work to rest time calculation
   RUNG wire#powerrail
      Contact( #DataOut.DrawHead.RestSolenoid )
      I_Contact( #Sts.CycleTime.DrawHead.W_To_R_Exe )
      { S7_Templates := "date_type := DTL" } RD_SYS_T(RET_VAL => #ReturnVal, OUT => #Sts.CycleTime.DrawHead.DT_R_Start)
      S_Coil( #Sts.CycleTime.DrawHead.W_To_R_Exe )
   END_RUNG
   RUNG wire#powerrail
      Contact( #Sts.CycleTime.DrawHead.W_To_R_Exe )
      wire#w1
      Contact( #PE.DrawHead.AtRest )
      wire#w2
      { S7_Templates := "date_type := DTL" } RD_SYS_T(RET_VAL => #ReturnVal, OUT => #Sts.CycleTime.DrawHead.DT_R_Stop)
   END_RUNG
   RUNG wire#w1
      I_Contact( #DataOut.DrawHead.RestSolenoid )
   END_RUNG wire#w2
   RUNG wire#w2
      { S7_Templates := "[date_type := DTL, time_type := Time]" } T_DIFF(IN1 := #Sts.CycleTime.DrawHead.DT_R_Stop, IN2 := #Sts.CycleTime.DrawHead.DT_R_Start, OUT => #HMI.DrawHead.Last_W_to_R_Time)
   END_RUNG
   RUNG wire#w2
      Add(in1 := #HMI.DrawHead.Buffer_W_to_R_Time[1].ID, in2 := 1, out => #HMI.DrawHead.Last_W_to_R_ID)
   END_RUNG
   RUNG wire#powerrail
      Contact( #Sts.CycleTime.DrawHead.W_To_R_Exe )
      I_Contact( #DataOut.DrawHead.RestSolenoid )
      R_Coil( #Sts.CycleTime.DrawHead.W_To_R_Exe )
   END_RUNG
   // the same network as SCL:
   #ReturnVal := RD_SYS_T(EN := #DataOut.DrawHead.RestSolenoid AND NOT #Sts.CycleTime.DrawHead.W_To_R_Exe,
                          OUT => #Sts.CycleTime.DrawHead.DT_R_Start,
                          ENO => #_w1);
   IF #_w1 THEN #Sts.CycleTime.DrawHead.W_To_R_Exe := TRUE; END_IF;
   IF #Sts.CycleTime.DrawHead.W_To_R_Exe AND (#PE.DrawHead.AtRest OR NOT #DataOut.DrawHead.RestSolenoid) THEN
       #ReturnVal := RD_SYS_T(OUT => #Sts.CycleTime.DrawHead.DT_R_Stop);
       T_DIFF(IN1 := #Sts.CycleTime.DrawHead.DT_R_Stop,
              IN2 := #Sts.CycleTime.DrawHead.DT_R_Start,
              OUT => #HMI.DrawHead.Last_W_to_R_Time);
       #HMI.DrawHead.Last_W_to_R_ID := #HMI.DrawHead.Buffer_W_to_R_Time[1].ID + 1;
   END_IF;
   IF #Sts.CycleTime.DrawHead.W_To_R_Exe AND NOT #DataOut.DrawHead.RestSolenoid THEN
       #Sts.CycleTime.DrawHead.W_To_R_Exe := FALSE;
   END_IF;
END_REGION

REGION Network 25 (SCL): Init buffers & average calculations
   IF #CIn.PPrf_PrgNo <> #Sts.CycleTime.PPrf_PrgNoSave OR #CIn.PPrf_PrgNo <= 0 THEN

       FOR #i := 1 TO #BUFFER_ITEMS DO
           #HMI.DrawHead.Buffer_R_to_W_Time[#i].ID := 0;
           #HMI.DrawHead.Buffer_R_to_W_Time[#i].Value := T#0s;
           #HMI.DrawHead.Buffer_W_to_R_Time[#i].ID := 0;
           #HMI.DrawHead.Buffer_W_to_R_Time[#i].Value := T#0s;
       END_FOR;

       #HMI.DrawHead.Last_R_to_W_ID := 0;
       #HMI.DrawHead.Last_R_to_W_Time := T#0ms;
       #HMI.DrawHead.Avg_R_to_W_Time := #Config.DrawHead.V.WorkTimeOut;

       #HMI.DrawHead.Last_W_to_R_ID := 0;
       #HMI.DrawHead.Last_W_to_R_Time := T#0ms;
       #HMI.DrawHead.Avg_W_to_R_Time := #Config.DrawHead.V.RestTimeOut;

   END_IF;


   #Sts.CycleTime.PPrf_PrgNoSave := #CIn.PPrf_PrgNo;
END_REGION

REGION Network 26 (SCL): Add new items to Rest-TO-Work buffer & calculate average

   IF #HMI.DrawHead.Last_R_to_W_Time >= #DrawHead.Config.V.WorkTimeOut OR #Alarm.DrawHead.TimeOutWork THEN

       #HMI.DrawHead.Last_R_to_W_ID := -1; // Force red background on the HMI visualization



   ELSIF #HMI.DrawHead.Last_R_to_W_ID <> #HMI.DrawHead.Buffer_R_to_W_Time[1].ID AND #HMI.DrawHead.Last_R_to_W_Time < #DrawHead.Config.V.WorkTimeOut AND #HMI.DrawHead.Last_R_to_W_Time > T#0ms THEN

       #i := #BUFFER_ITEMS;

       WHILE #i >= 2 DO

           #HMI.DrawHead.Buffer_R_to_W_Time[#i] := #HMI.DrawHead.Buffer_R_to_W_Time[#i - 1];

           #i -= 1;

       END_WHILE;

       #HMI.DrawHead.Buffer_R_to_W_Time[1].ID := #HMI.DrawHead.Last_R_to_W_ID;
       #HMI.DrawHead.Buffer_R_to_W_Time[1].Value := #HMI.DrawHead.Last_R_to_W_Time;

       #Sts.CycleTime.DrawHead.R_To_W_Items := 0;
       #Sts.CycleTime.DrawHead.R_To_W_Sum := T#0s;


       FOR #i := 1 TO #BUFFER_ITEMS DO

           IF #HMI.DrawHead.Buffer_R_to_W_Time[#i].ID > 0 AND #HMI.DrawHead.Buffer_R_to_W_Time[#i].Value > T#0ms THEN
               #Sts.CycleTime.DrawHead.R_To_W_Items += 1;
               #Sts.CycleTime.DrawHead.R_To_W_Sum := #Sts.CycleTime.DrawHead.R_To_W_Sum + #HMI.DrawHead.Buffer_R_to_W_Time[#i].Value;
           END_IF;

       END_FOR;

       IF #Sts.CycleTime.DrawHead.R_To_W_Items >= 5 THEN
           #HMI.DrawHead.Avg_R_to_W_Time := #Sts.CycleTime.DrawHead.R_To_W_Sum / #Sts.CycleTime.DrawHead.R_To_W_Items;
       ELSE
           #HMI.DrawHead.Avg_R_to_W_Time := #Config.DrawHead.V.WorkTimeOut;
       END_IF;

   END_IF;
END_REGION

REGION Network 27 (SCL): Add new items to Work-TO-Rest buffer & calculate average
   IF #HMI.DrawHead.Last_W_to_R_Time >= #DrawHead.Config.V.RestTimeOut OR #Alarm.DrawHead.TimeOutRest THEN

       #HMI.DrawHead.Last_W_to_R_ID := -1; // Force red background on the HMI visualization

   ELSIF #HMI.DrawHead.Last_W_to_R_ID <> #HMI.DrawHead.Buffer_W_to_R_Time[1].ID AND #HMI.DrawHead.Last_W_to_R_Time < #DrawHead.Config.V.RestTimeOut AND #HMI.DrawHead.Last_W_to_R_Time > T#0ms  THEN

       #i := #BUFFER_ITEMS;

       WHILE #i >= 2 DO

           #HMI.DrawHead.Buffer_W_to_R_Time[#i] := #HMI.DrawHead.Buffer_W_to_R_Time[#i - 1];

           #i -= 1;

       END_WHILE;

       #HMI.DrawHead.Buffer_W_to_R_Time[1].ID := #HMI.DrawHead.Last_W_to_R_ID;
       #HMI.DrawHead.Buffer_W_to_R_Time[1].Value := #HMI.DrawHead.Last_W_to_R_Time;

       #Sts.CycleTime.DrawHead.W_To_R_Items := 0;
       #Sts.CycleTime.DrawHead.W_To_R_Sum := T#0s;


       FOR #i := 1 TO #BUFFER_ITEMS DO

           IF #HMI.DrawHead.Buffer_W_to_R_Time[#i].ID > 0 AND #HMI.DrawHead.Buffer_W_to_R_Time[#i].Value > T#0ms  THEN
               #Sts.CycleTime.DrawHead.W_To_R_Items += 1;
               #Sts.CycleTime.DrawHead.W_To_R_Sum := #Sts.CycleTime.DrawHead.W_To_R_Sum + #HMI.DrawHead.Buffer_W_to_R_Time[#i].Value;
           END_IF;

       END_FOR;

       IF #Sts.CycleTime.DrawHead.W_To_R_Items >= 5 THEN
           #HMI.DrawHead.Avg_W_to_R_Time := #Sts.CycleTime.DrawHead.W_To_R_Sum / #Sts.CycleTime.DrawHead.W_To_R_Items;
       ELSE
           #HMI.DrawHead.Avg_W_to_R_Time := #Config.DrawHead.V.RestTimeOut;
       END_IF;

   END_IF;
END_REGION

REGION Network 28: >
END_REGION

REGION Network 29: <<< MARKING HEAD >>>
END_REGION

REGION Network 30: Pressure reload for avoiding losing of rest position cause leakage on hydraulic cylinders
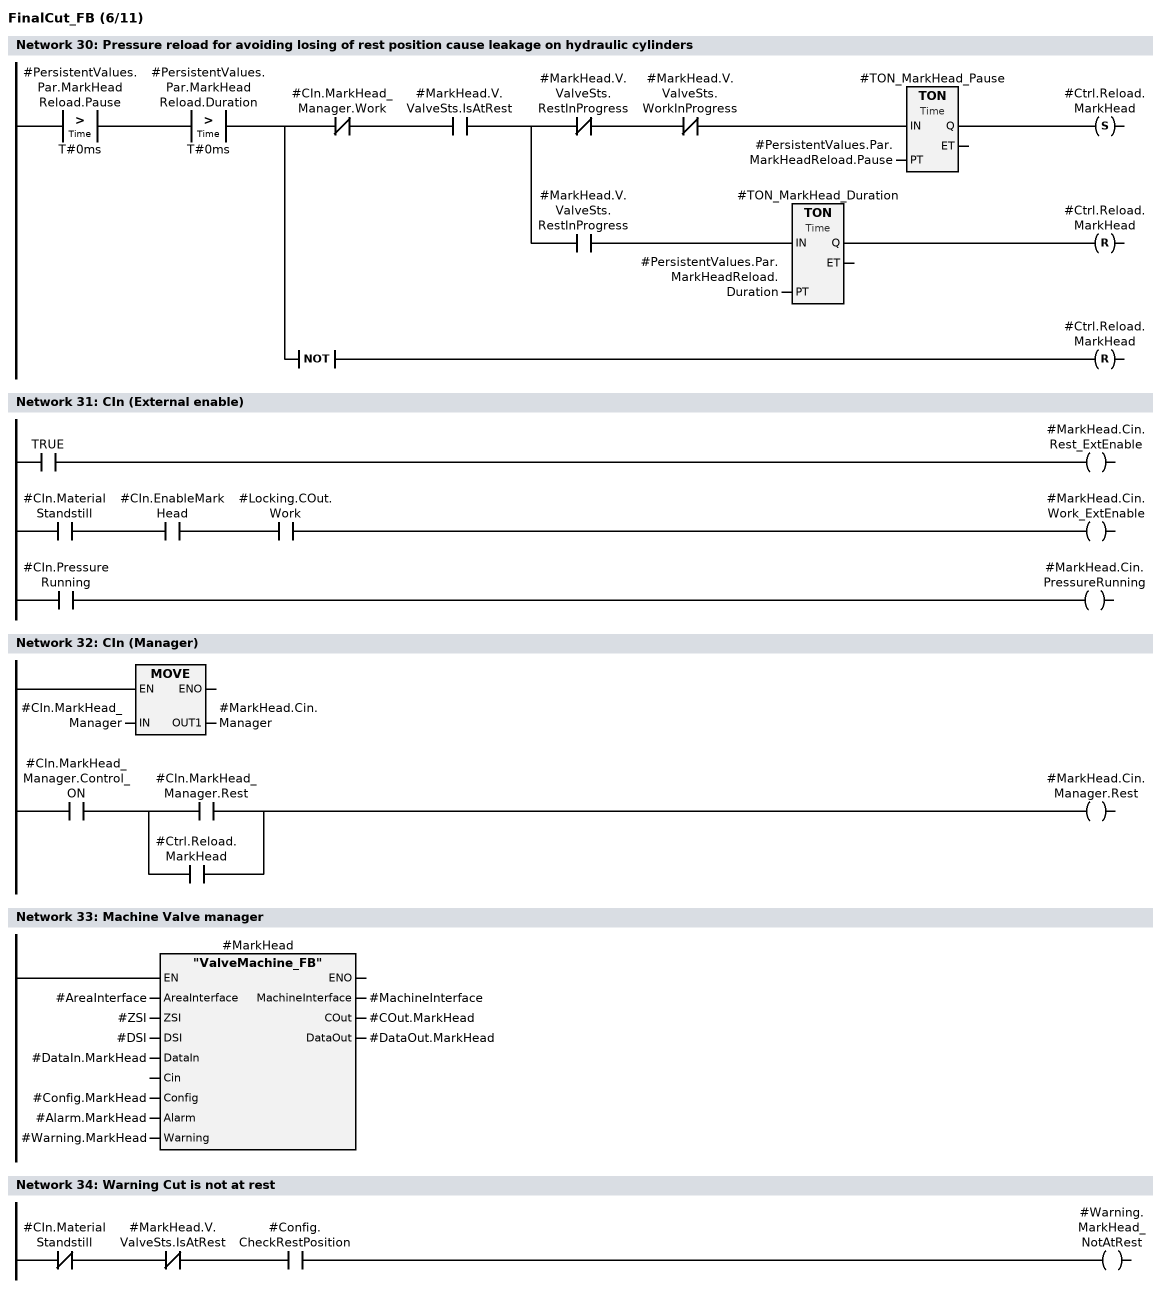
   RUNG wire#powerrail
      { S7_Templates := "SrcType := Time" } GT_Contact(in1 := #PersistentValues.Par.MarkHeadReload.Pause, in2 := T#0ms)
      { S7_Templates := "SrcType := Time" } GT_Contact(in1 := #PersistentValues.Par.MarkHeadReload.Duration, in2 := T#0ms)
      wire#w1
      I_Contact( #CIn.MarkHead_Manager.Work )
      Contact( #MarkHead.V.ValveSts.IsAtRest )
      wire#w2
      I_Contact( #MarkHead.V.ValveSts.RestInProgress )
      I_Contact( #MarkHead.V.ValveSts.WorkInProgress )
      { S7_Templates := "time_type := Time" } #TON_MarkHead_Pause.TON(pt := #PersistentValues.Par.MarkHeadReload.Pause, et =>)
      S_Coil( #Ctrl.Reload.MarkHead )
   END_RUNG
   RUNG wire#w2
      Contact( #MarkHead.V.ValveSts.RestInProgress )
      { S7_Templates := "time_type := Time" } #TON_MarkHead_Duration.TON(pt := #PersistentValues.Par.MarkHeadReload.Duration, et =>)
      R_Coil( #Ctrl.Reload.MarkHead )
   END_RUNG
   RUNG wire#w1
      Not()
      R_Coil( #Ctrl.Reload.MarkHead )
   END_RUNG
   // the same network as SCL:
   #_w1 := (#PersistentValues.Par.MarkHeadReload.Pause > T#0ms) AND (#PersistentValues.Par.MarkHeadReload.Duration > T#0ms);
   #_w2 := #_w1 AND NOT #CIn.MarkHead_Manager.Work AND #MarkHead.V.ValveSts.IsAtRest;
   #TON_MarkHead_Pause.TON(IN := #_w2 AND NOT #MarkHead.V.ValveSts.RestInProgress AND NOT #MarkHead.V.ValveSts.WorkInProgress,
                           PT := #PersistentValues.Par.MarkHeadReload.Pause);
   IF #TON_MarkHead_Pause.Q THEN #Ctrl.Reload.MarkHead := TRUE; END_IF;
   #TON_MarkHead_Duration.TON(IN := #_w2 AND #MarkHead.V.ValveSts.RestInProgress,
                           PT := #PersistentValues.Par.MarkHeadReload.Duration);
   IF #TON_MarkHead_Duration.Q THEN #Ctrl.Reload.MarkHead := FALSE; END_IF;
   IF NOT #_w1 THEN #Ctrl.Reload.MarkHead := FALSE; END_IF;
END_REGION

REGION Network 31: CIn (External enable)
   RUNG wire#powerrail
      Contact( TRUE )
      Coil( #MarkHead.Cin.Rest_ExtEnable )
   END_RUNG
   RUNG wire#powerrail
      Contact( #CIn.MaterialStandstill )
      Contact( #CIn.EnableMarkHead )
      Contact( #Locking.COut.Work )
      Coil( #MarkHead.Cin.Work_ExtEnable )
   END_RUNG
   RUNG wire#powerrail
      Contact( #CIn.PressureRunning )
      Coil( #MarkHead.Cin.PressureRunning )
   END_RUNG
   // the same network as SCL:
   #MarkHead.Cin.Rest_ExtEnable := TRUE;
   #MarkHead.Cin.Work_ExtEnable := #CIn.MaterialStandstill AND #CIn.EnableMarkHead AND #Locking.COut.Work;
   #MarkHead.Cin.PressureRunning := #CIn.PressureRunning;
END_REGION

REGION Network 32: CIn (Manager)
   RUNG wire#powerrail
      Move(in := #CIn.MarkHead_Manager, out1 => #MarkHead.Cin.Manager)
   END_RUNG
   RUNG wire#powerrail
      Contact( #CIn.MarkHead_Manager.Control_ON )
      wire#w1
      Contact( #CIn.MarkHead_Manager.Rest )
      wire#w2
      Coil( #MarkHead.Cin.Manager.Rest )
   END_RUNG
   RUNG wire#w1
      Contact( #Ctrl.Reload.MarkHead )
   END_RUNG wire#w2
   // the same network as SCL:
   #MarkHead.Cin.Manager := #CIn.MarkHead_Manager;
   #MarkHead.Cin.Manager.Rest := #CIn.MarkHead_Manager.Control_ON AND (#CIn.MarkHead_Manager.Rest OR #Ctrl.Reload.MarkHead);
END_REGION

REGION Network 33: Machine Valve manager
   RUNG wire#powerrail
      #MarkHead(AreaInterface := #AreaInterface, ZSI := #ZSI, DSI := #DSI, DataIn := #DataIn.MarkHead, Cin :=, Config := #Config.MarkHead, Alarm := #Alarm.MarkHead, Warning := #Warning.MarkHead, MachineInterface => #MachineInterface, COut => #COut.MarkHead, DataOut => #DataOut.MarkHead)
   END_RUNG
   // the same network as SCL:
   #MarkHead(AreaInterface := #AreaInterface,   // "ValveMachine_FB"
             ZSI := #ZSI,
             DSI := #DSI,
             DataIn := #DataIn.MarkHead,
             Config := #Config.MarkHead,
             Alarm := #Alarm.MarkHead,
             Warning := #Warning.MarkHead,
             MachineInterface => #MachineInterface,
             COut => #COut.MarkHead,
             DataOut => #DataOut.MarkHead);
END_REGION

REGION Network 34: Warning Cut is not at rest
   RUNG wire#powerrail
      I_Contact( #CIn.MaterialStandstill )
      I_Contact( #MarkHead.V.ValveSts.IsAtRest )
      Contact( #Config.CheckRestPosition )
      Coil( #Warning.MarkHead_NotAtRest )
   END_RUNG
   // the same network as SCL:
   #Warning.MarkHead_NotAtRest := NOT #CIn.MaterialStandstill AND NOT #MarkHead.V.ValveSts.IsAtRest AND #Config.CheckRestPosition;
END_REGION

REGION Network 35: At Rest / At work positive/negative edge
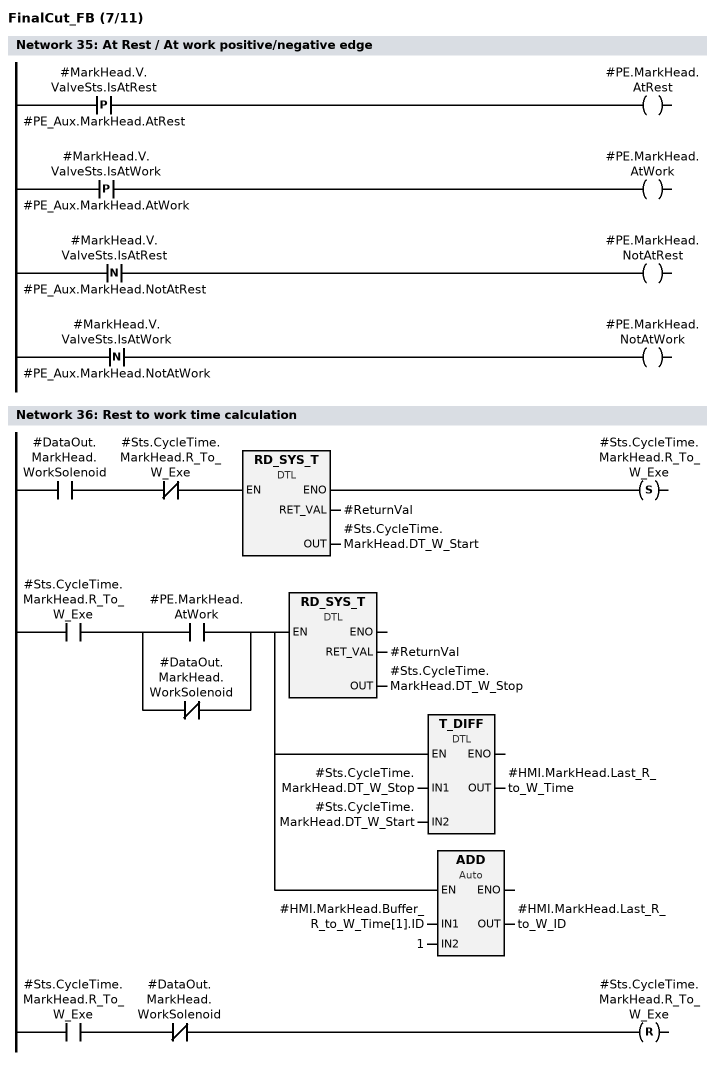
   RUNG wire#powerrail
      P_Contact(operand := #MarkHead.V.ValveSts.IsAtRest, bit := #PE_Aux.MarkHead.AtRest)
      Coil( #PE.MarkHead.AtRest )
   END_RUNG
   RUNG wire#powerrail
      P_Contact(operand := #MarkHead.V.ValveSts.IsAtWork, bit := #PE_Aux.MarkHead.AtWork)
      Coil( #PE.MarkHead.AtWork )
   END_RUNG
   RUNG wire#powerrail
      N_Contact(operand := #MarkHead.V.ValveSts.IsAtRest, bit := #PE_Aux.MarkHead.NotAtRest)
      Coil( #PE.MarkHead.NotAtRest )
   END_RUNG
   RUNG wire#powerrail
      N_Contact(operand := #MarkHead.V.ValveSts.IsAtWork, bit := #PE_Aux.MarkHead.NotAtWork)
      Coil( #PE.MarkHead.NotAtWork )
   END_RUNG
   // the same network as SCL:
   #_w1 := #MarkHead.V.ValveSts.IsAtRest AND NOT #PE_Aux.MarkHead.AtRest;   // rising edge of #MarkHead.V.ValveSts.IsAtRest
   #PE_Aux.MarkHead.AtRest := #MarkHead.V.ValveSts.IsAtRest;
   #PE.MarkHead.AtRest := #_w1;
   #_w2 := #MarkHead.V.ValveSts.IsAtWork AND NOT #PE_Aux.MarkHead.AtWork;   // rising edge of #MarkHead.V.ValveSts.IsAtWork
   #PE_Aux.MarkHead.AtWork := #MarkHead.V.ValveSts.IsAtWork;
   #PE.MarkHead.AtWork := #_w2;
   #_w3 := NOT #MarkHead.V.ValveSts.IsAtRest AND #PE_Aux.MarkHead.NotAtRest;   // falling edge of #MarkHead.V.ValveSts.IsAtRest
   #PE_Aux.MarkHead.NotAtRest := #MarkHead.V.ValveSts.IsAtRest;
   #PE.MarkHead.NotAtRest := #_w3;
   #_w4 := NOT #MarkHead.V.ValveSts.IsAtWork AND #PE_Aux.MarkHead.NotAtWork;   // falling edge of #MarkHead.V.ValveSts.IsAtWork
   #PE_Aux.MarkHead.NotAtWork := #MarkHead.V.ValveSts.IsAtWork;
   #PE.MarkHead.NotAtWork := #_w4;
END_REGION

REGION Network 36: Rest to work time calculation
   RUNG wire#powerrail
      Contact( #DataOut.MarkHead.WorkSolenoid )
      I_Contact( #Sts.CycleTime.MarkHead.R_To_W_Exe )
      { S7_Templates := "date_type := DTL" } RD_SYS_T(RET_VAL => #ReturnVal, OUT => #Sts.CycleTime.MarkHead.DT_W_Start)
      S_Coil( #Sts.CycleTime.MarkHead.R_To_W_Exe )
   END_RUNG
   RUNG wire#powerrail
      Contact( #Sts.CycleTime.MarkHead.R_To_W_Exe )
      wire#w1
      Contact( #PE.MarkHead.AtWork )
      wire#w2
      { S7_Templates := "date_type := DTL" } RD_SYS_T(RET_VAL => #ReturnVal, OUT => #Sts.CycleTime.MarkHead.DT_W_Stop)
   END_RUNG
   RUNG wire#w1
      I_Contact( #DataOut.MarkHead.WorkSolenoid )
   END_RUNG wire#w2
   RUNG wire#w2
      { S7_Templates := "[date_type := DTL, time_type := Time]" } T_DIFF(IN1 := #Sts.CycleTime.MarkHead.DT_W_Stop, IN2 := #Sts.CycleTime.MarkHead.DT_W_Start, OUT => #HMI.MarkHead.Last_R_to_W_Time)
   END_RUNG
   RUNG wire#w2
      Add(in1 := #HMI.MarkHead.Buffer_R_to_W_Time[1].ID, in2 := 1, out => #HMI.MarkHead.Last_R_to_W_ID)
   END_RUNG
   RUNG wire#powerrail
      Contact( #Sts.CycleTime.MarkHead.R_To_W_Exe )
      I_Contact( #DataOut.MarkHead.WorkSolenoid )
      R_Coil( #Sts.CycleTime.MarkHead.R_To_W_Exe )
   END_RUNG
   // the same network as SCL:
   #ReturnVal := RD_SYS_T(EN := #DataOut.MarkHead.WorkSolenoid AND NOT #Sts.CycleTime.MarkHead.R_To_W_Exe,
                          OUT => #Sts.CycleTime.MarkHead.DT_W_Start,
                          ENO => #_w1);
   IF #_w1 THEN #Sts.CycleTime.MarkHead.R_To_W_Exe := TRUE; END_IF;
   IF #Sts.CycleTime.MarkHead.R_To_W_Exe AND (#PE.MarkHead.AtWork OR NOT #DataOut.MarkHead.WorkSolenoid) THEN
       #ReturnVal := RD_SYS_T(OUT => #Sts.CycleTime.MarkHead.DT_W_Stop);
       T_DIFF(IN1 := #Sts.CycleTime.MarkHead.DT_W_Stop,
              IN2 := #Sts.CycleTime.MarkHead.DT_W_Start,
              OUT => #HMI.MarkHead.Last_R_to_W_Time);
       #HMI.MarkHead.Last_R_to_W_ID := #HMI.MarkHead.Buffer_R_to_W_Time[1].ID + 1;
   END_IF;
   IF #Sts.CycleTime.MarkHead.R_To_W_Exe AND NOT #DataOut.MarkHead.WorkSolenoid THEN
       #Sts.CycleTime.MarkHead.R_To_W_Exe := FALSE;
   END_IF;
END_REGION

REGION Network 37: Work to rest time calculation
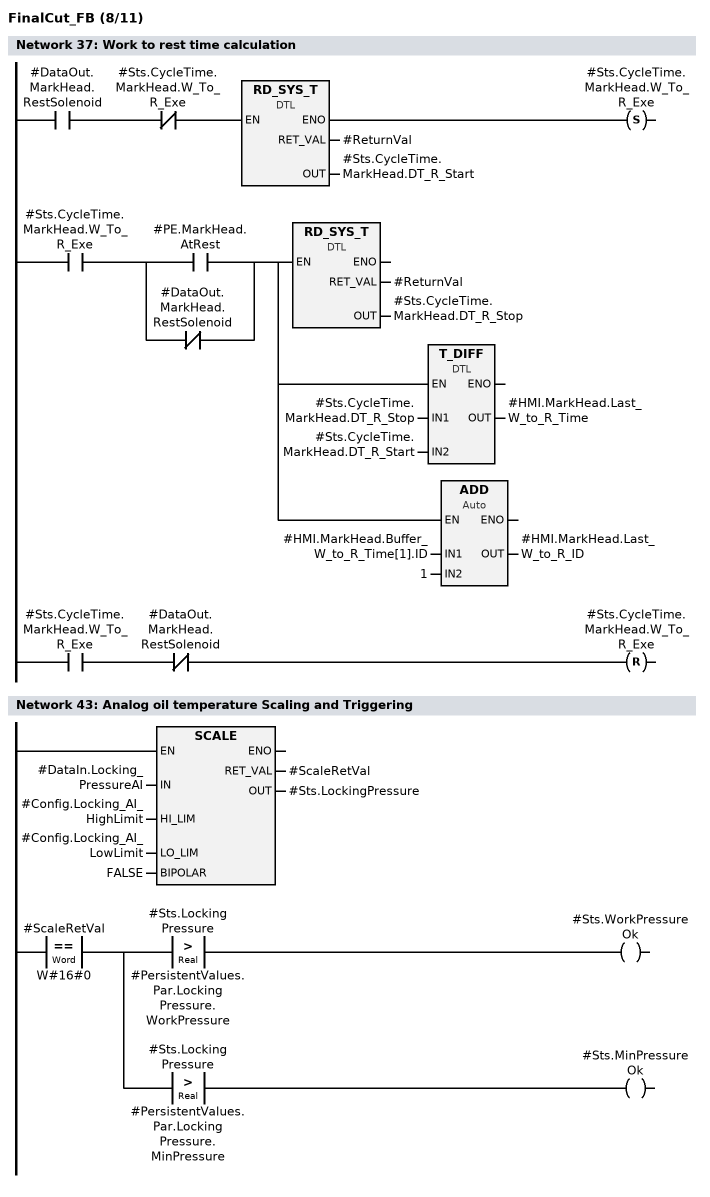
   RUNG wire#powerrail
      Contact( #DataOut.MarkHead.RestSolenoid )
      I_Contact( #Sts.CycleTime.MarkHead.W_To_R_Exe )
      { S7_Templates := "date_type := DTL" } RD_SYS_T(RET_VAL => #ReturnVal, OUT => #Sts.CycleTime.MarkHead.DT_R_Start)
      S_Coil( #Sts.CycleTime.MarkHead.W_To_R_Exe )
   END_RUNG
   RUNG wire#powerrail
      Contact( #Sts.CycleTime.MarkHead.W_To_R_Exe )
      wire#w1
      Contact( #PE.MarkHead.AtRest )
      wire#w2
      { S7_Templates := "date_type := DTL" } RD_SYS_T(RET_VAL => #ReturnVal, OUT => #Sts.CycleTime.MarkHead.DT_R_Stop)
   END_RUNG
   RUNG wire#w1
      I_Contact( #DataOut.MarkHead.RestSolenoid )
   END_RUNG wire#w2
   RUNG wire#w2
      { S7_Templates := "[date_type := DTL, time_type := Time]" } T_DIFF(IN1 := #Sts.CycleTime.MarkHead.DT_R_Stop, IN2 := #Sts.CycleTime.MarkHead.DT_R_Start, OUT => #HMI.MarkHead.Last_W_to_R_Time)
   END_RUNG
   RUNG wire#w2
      Add(in1 := #HMI.MarkHead.Buffer_W_to_R_Time[1].ID, in2 := 1, out => #HMI.MarkHead.Last_W_to_R_ID)
   END_RUNG
   RUNG wire#powerrail
      Contact( #Sts.CycleTime.MarkHead.W_To_R_Exe )
      I_Contact( #DataOut.MarkHead.RestSolenoid )
      R_Coil( #Sts.CycleTime.MarkHead.W_To_R_Exe )
   END_RUNG
   // the same network as SCL:
   #ReturnVal := RD_SYS_T(EN := #DataOut.MarkHead.RestSolenoid AND NOT #Sts.CycleTime.MarkHead.W_To_R_Exe,
                          OUT => #Sts.CycleTime.MarkHead.DT_R_Start,
                          ENO => #_w1);
   IF #_w1 THEN #Sts.CycleTime.MarkHead.W_To_R_Exe := TRUE; END_IF;
   IF #Sts.CycleTime.MarkHead.W_To_R_Exe AND (#PE.MarkHead.AtRest OR NOT #DataOut.MarkHead.RestSolenoid) THEN
       #ReturnVal := RD_SYS_T(OUT => #Sts.CycleTime.MarkHead.DT_R_Stop);
       T_DIFF(IN1 := #Sts.CycleTime.MarkHead.DT_R_Stop,
              IN2 := #Sts.CycleTime.MarkHead.DT_R_Start,
              OUT => #HMI.MarkHead.Last_W_to_R_Time);
       #HMI.MarkHead.Last_W_to_R_ID := #HMI.MarkHead.Buffer_W_to_R_Time[1].ID + 1;
   END_IF;
   IF #Sts.CycleTime.MarkHead.W_To_R_Exe AND NOT #DataOut.MarkHead.RestSolenoid THEN
       #Sts.CycleTime.MarkHead.W_To_R_Exe := FALSE;
   END_IF;
END_REGION

REGION Network 38 (SCL): Init buffers & average calculations
   IF #CIn.PPrf_PrgNo <> #Sts.CycleTime.PPrf_PrgNoSave OR #CIn.PPrf_PrgNo <= 0 THEN

       FOR #i := 1 TO #BUFFER_ITEMS DO
           #HMI.MarkHead.Buffer_R_to_W_Time[#i].ID := 0;
           #HMI.MarkHead.Buffer_R_to_W_Time[#i].Value := T#0s;
           #HMI.MarkHead.Buffer_W_to_R_Time[#i].ID := 0;
           #HMI.MarkHead.Buffer_W_to_R_Time[#i].Value := T#0s;
       END_FOR;

       #HMI.MarkHead.Last_R_to_W_ID := 0;
       #HMI.MarkHead.Last_R_to_W_Time := T#0ms;
       #HMI.MarkHead.Avg_R_to_W_Time := #Config.MarkHead.V.WorkTimeOut;

       #HMI.MarkHead.Last_W_to_R_ID := 0;
       #HMI.MarkHead.Last_W_to_R_Time := T#0ms;
       #HMI.MarkHead.Avg_W_to_R_Time := #Config.MarkHead.V.RestTimeOut;

   END_IF;


   #Sts.CycleTime.PPrf_PrgNoSave := #CIn.PPrf_PrgNo;
END_REGION

REGION Network 39 (SCL): Add new items to Rest-TO-Work buffer & calculate average

   IF #HMI.MarkHead.Last_R_to_W_Time >= #MarkHead.Config.V.WorkTimeOut OR #Alarm.MarkHead.TimeOutWork THEN

       #HMI.MarkHead.Last_R_to_W_ID := -1; // Force red background on the HMI visualization



   ELSIF #HMI.MarkHead.Last_R_to_W_ID <> #HMI.MarkHead.Buffer_R_to_W_Time[1].ID AND #HMI.MarkHead.Last_R_to_W_Time < #MarkHead.Config.V.WorkTimeOut AND #HMI.MarkHead.Last_R_to_W_Time > T#0ms THEN

       #i := #BUFFER_ITEMS;

       WHILE #i >= 2 DO

           #HMI.MarkHead.Buffer_R_to_W_Time[#i] := #HMI.MarkHead.Buffer_R_to_W_Time[#i - 1];

           #i -= 1;

       END_WHILE;

       #HMI.MarkHead.Buffer_R_to_W_Time[1].ID := #HMI.MarkHead.Last_R_to_W_ID;
       #HMI.MarkHead.Buffer_R_to_W_Time[1].Value := #HMI.MarkHead.Last_R_to_W_Time;

       #Sts.CycleTime.MarkHead.R_To_W_Items := 0;
       #Sts.CycleTime.MarkHead.R_To_W_Sum := T#0s;


       FOR #i := 1 TO #BUFFER_ITEMS DO

           IF #HMI.MarkHead.Buffer_R_to_W_Time[#i].ID > 0 AND #HMI.MarkHead.Buffer_R_to_W_Time[#i].Value > T#0ms THEN
               #Sts.CycleTime.MarkHead.R_To_W_Items += 1;
               #Sts.CycleTime.MarkHead.R_To_W_Sum := #Sts.CycleTime.MarkHead.R_To_W_Sum + #HMI.MarkHead.Buffer_R_to_W_Time[#i].Value;
           END_IF;

       END_FOR;

       IF #Sts.CycleTime.MarkHead.R_To_W_Items >= 5 THEN
           #HMI.MarkHead.Avg_R_to_W_Time := #Sts.CycleTime.MarkHead.R_To_W_Sum / #Sts.CycleTime.MarkHead.R_To_W_Items;
       ELSE
           #HMI.MarkHead.Avg_R_to_W_Time := #Config.MarkHead.V.WorkTimeOut;
       END_IF;

   END_IF;
END_REGION

REGION Network 40 (SCL): Add new items to Work-TO-Rest buffer & calculate average
   IF #HMI.MarkHead.Last_W_to_R_Time >= #MarkHead.Config.V.RestTimeOut OR #Alarm.MarkHead.TimeOutRest THEN

       #HMI.MarkHead.Last_W_to_R_ID := -1; // Force red background on the HMI visualization

   ELSIF #HMI.MarkHead.Last_W_to_R_ID <> #HMI.MarkHead.Buffer_W_to_R_Time[1].ID AND #HMI.MarkHead.Last_W_to_R_Time < #MarkHead.Config.V.RestTimeOut AND #HMI.MarkHead.Last_W_to_R_Time > T#0ms  THEN

       #i := #BUFFER_ITEMS;

       WHILE #i >= 2 DO

           #HMI.MarkHead.Buffer_W_to_R_Time[#i] := #HMI.MarkHead.Buffer_W_to_R_Time[#i - 1];

           #i -= 1;

       END_WHILE;

       #HMI.MarkHead.Buffer_W_to_R_Time[1].ID := #HMI.MarkHead.Last_W_to_R_ID;
       #HMI.MarkHead.Buffer_W_to_R_Time[1].Value := #HMI.MarkHead.Last_W_to_R_Time;

       #Sts.CycleTime.MarkHead.W_To_R_Items := 0;
       #Sts.CycleTime.MarkHead.W_To_R_Sum := T#0s;


       FOR #i := 1 TO #BUFFER_ITEMS DO

           IF #HMI.MarkHead.Buffer_W_to_R_Time[#i].ID > 0 AND #HMI.MarkHead.Buffer_W_to_R_Time[#i].Value > T#0ms  THEN
               #Sts.CycleTime.MarkHead.W_To_R_Items += 1;
               #Sts.CycleTime.MarkHead.W_To_R_Sum := #Sts.CycleTime.MarkHead.W_To_R_Sum + #HMI.MarkHead.Buffer_W_to_R_Time[#i].Value;
           END_IF;

       END_FOR;

       IF #Sts.CycleTime.MarkHead.W_To_R_Items >= 5 THEN
           #HMI.MarkHead.Avg_W_to_R_Time := #Sts.CycleTime.MarkHead.W_To_R_Sum / #Sts.CycleTime.MarkHead.W_To_R_Items;
       ELSE
           #HMI.MarkHead.Avg_W_to_R_Time := #Config.MarkHead.V.RestTimeOut;
       END_IF;

   END_IF;
END_REGION

REGION Network 41: >
END_REGION

REGION Network 42: <<< LOCKING >>>
END_REGION

REGION Network 43: Analog oil temperature Scaling and Triggering
   #ScaleRetVal := SCALE(IN := #DataIn.Locking_PressureAI,
                         HI_LIM := #Config.Locking_AI_HighLimit,
                         LO_LIM := #Config.Locking_AI_LowLimit,
                         BIPOLAR := FALSE,
                         OUT => #Sts.LockingPressure);
   #_w1 := #ScaleRetVal = W#16#0;
   #Sts.WorkPressureOk := #_w1 AND (#Sts.LockingPressure > #PersistentValues.Par.LockingPressure.WorkPressure);
   #Sts.MinPressureOk := #_w1 AND (#Sts.LockingPressure > #PersistentValues.Par.LockingPressure.MinPressure);
END_REGION

REGION Network 44: Pressure reload for avoiding losing of rest position cause leakage on hydraulic cylinders
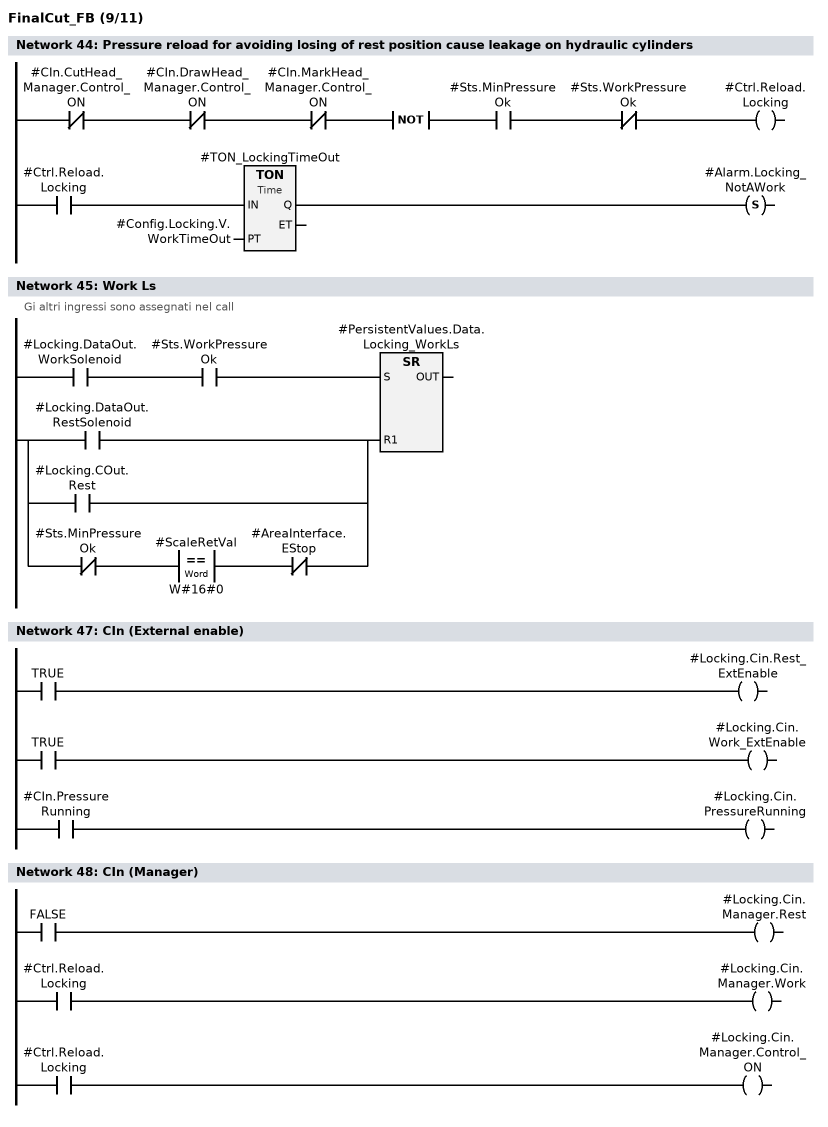
   RUNG wire#powerrail
      I_Contact( #CIn.CutHead_Manager.Control_ON )
      I_Contact( #CIn.DrawHead_Manager.Control_ON )
      I_Contact( #CIn.MarkHead_Manager.Control_ON )
      Not()
      Contact( #Sts.MinPressureOk )
      I_Contact( #Sts.WorkPressureOk )
      Coil( #Ctrl.Reload.Locking )
   END_RUNG
   RUNG wire#powerrail
      Contact( #Ctrl.Reload.Locking )
      { S7_Templates := "time_type := Time" } #TON_LockingTimeOut.TON(pt := #Config.Locking.V.WorkTimeOut, et =>)
      S_Coil( #Alarm.Locking_NotAWork )
   END_RUNG
   // the same network as SCL:
   #Ctrl.Reload.Locking := NOT (NOT #CIn.CutHead_Manager.Control_ON AND NOT #CIn.DrawHead_Manager.Control_ON AND NOT #CIn.MarkHead_Manager.Control_ON) AND #Sts.MinPressureOk AND NOT #Sts.WorkPressureOk;
   #TON_LockingTimeOut.TON(IN := #Ctrl.Reload.Locking, PT := #Config.Locking.V.WorkTimeOut);
   IF #TON_LockingTimeOut.Q THEN #Alarm.Locking_NotAWork := TRUE; END_IF;
END_REGION

REGION Network 45: Work Ls
   // Gi altri ingressi sono assegnati nel call
   RUNG wire#powerrail
      Contact( #Locking.DataOut.WorkSolenoid )
      Contact( #Sts.WorkPressureOk )
      S_SR(operand := #PersistentValues.Data.Locking_WorkLs, r1 := wire#w1)
   END_RUNG
   RUNG wire#powerrail
      Contact( #Locking.DataOut.RestSolenoid )
   END_RUNG wire#w1
   RUNG wire#powerrail
      Contact( #Locking.COut.Rest )
   END_RUNG wire#w1
   RUNG wire#powerrail
      I_Contact( #Sts.MinPressureOk )
      { S7_Templates := "SrcType := Word" } EQ_Contact(in1 := #ScaleRetVal, in2 := W#16#0)
      I_Contact( #AreaInterface.EStop )
   END_RUNG wire#w1
   // the same network as SCL:
   IF #Locking.DataOut.WorkSolenoid AND #Sts.WorkPressureOk THEN
       #PersistentValues.Data.Locking_WorkLs := TRUE;   // SR flip-flop
   END_IF;
   IF #Locking.DataOut.RestSolenoid OR #Locking.COut.Rest OR (NOT #Sts.MinPressureOk AND (#ScaleRetVal = W#16#0) AND NOT #AreaInterface.EStop) THEN
       #PersistentValues.Data.Locking_WorkLs := FALSE;
   END_IF;
END_REGION

REGION Network 46 (SCL): Data In
   #Locking.DataIn := #DataIn.Locking;

   #Locking.DataIn.Work_Ls[1] := #PersistentValues.Data.Locking_WorkLs;
END_REGION

REGION Network 47: CIn (External enable)
   RUNG wire#powerrail
      Contact( TRUE )
      Coil( #Locking.Cin.Rest_ExtEnable )
   END_RUNG
   RUNG wire#powerrail
      Contact( TRUE )
      Coil( #Locking.Cin.Work_ExtEnable )
   END_RUNG
   RUNG wire#powerrail
      Contact( #CIn.PressureRunning )
      Coil( #Locking.Cin.PressureRunning )
   END_RUNG
   // the same network as SCL:
   #Locking.Cin.Rest_ExtEnable := TRUE;
   #Locking.Cin.Work_ExtEnable := TRUE;
   #Locking.Cin.PressureRunning := #CIn.PressureRunning;
END_REGION

REGION Network 48: CIn (Manager)
   RUNG wire#powerrail
      Contact( FALSE )
      Coil( #Locking.Cin.Manager.Rest )
   END_RUNG
   RUNG wire#powerrail
      Contact( #Ctrl.Reload.Locking )
      Coil( #Locking.Cin.Manager.Work )
   END_RUNG
   RUNG wire#powerrail
      Contact( #Ctrl.Reload.Locking )
      Coil( #Locking.Cin.Manager.Control_ON )
   END_RUNG
   // the same network as SCL:
   #Locking.Cin.Manager.Rest := FALSE;
   #Locking.Cin.Manager.Work := #Ctrl.Reload.Locking;
   #Locking.Cin.Manager.Control_ON := #Ctrl.Reload.Locking;
END_REGION

REGION Network 49: Machine Valve manager
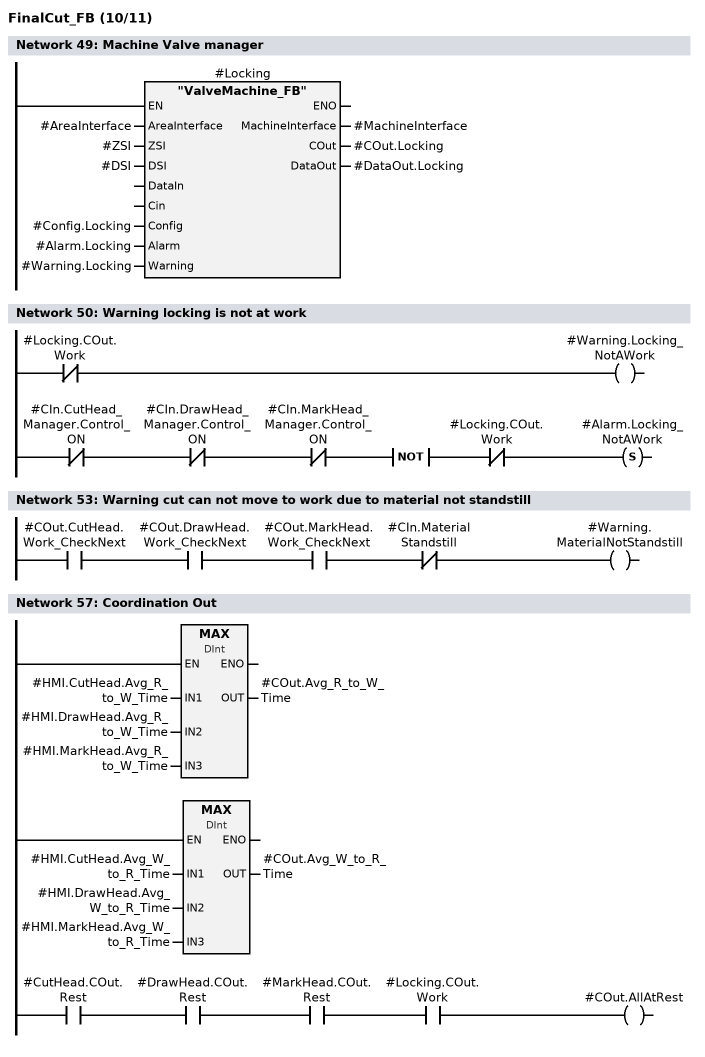
   RUNG wire#powerrail
      #Locking(AreaInterface := #AreaInterface, ZSI := #ZSI, DSI := #DSI, DataIn :=, Cin :=, Config := #Config.Locking, Alarm := #Alarm.Locking, Warning := #Warning.Locking, MachineInterface => #MachineInterface, COut => #COut.Locking, DataOut => #DataOut.Locking)
   END_RUNG
   // the same network as SCL:
   #Locking(AreaInterface := #AreaInterface,   // "ValveMachine_FB"
            ZSI := #ZSI,
            DSI := #DSI,
            Config := #Config.Locking,
            Alarm := #Alarm.Locking,
            Warning := #Warning.Locking,
            MachineInterface => #MachineInterface,
            COut => #COut.Locking,
            DataOut => #DataOut.Locking);
END_REGION

REGION Network 50: Warning locking is not at work
   RUNG wire#powerrail
      I_Contact( #Locking.COut.Work )
      Coil( #Warning.Locking_NotAWork )
   END_RUNG
   RUNG wire#powerrail
      I_Contact( #CIn.CutHead_Manager.Control_ON )
      I_Contact( #CIn.DrawHead_Manager.Control_ON )
      I_Contact( #CIn.MarkHead_Manager.Control_ON )
      Not()
      I_Contact( #Locking.COut.Work )
      S_Coil( #Alarm.Locking_NotAWork )
   END_RUNG
   // the same network as SCL:
   #Warning.Locking_NotAWork := NOT #Locking.COut.Work;
   IF NOT (NOT #CIn.CutHead_Manager.Control_ON AND NOT #CIn.DrawHead_Manager.Control_ON AND NOT #CIn.MarkHead_Manager.Control_ON) AND NOT #Locking.COut.Work THEN
       #Alarm.Locking_NotAWork := TRUE;
   END_IF;
END_REGION

REGION Network 51: >
END_REGION

REGION Network 52: <<< MISCELLANEUS>>>
END_REGION

REGION Network 53: Warning cut can not move to work due to material not standstill
   RUNG wire#powerrail
      Contact( #COut.CutHead.Work_CheckNext )
      Contact( #COut.DrawHead.Work_CheckNext )
      Contact( #COut.MarkHead.Work_CheckNext )
      I_Contact( #CIn.MaterialStandstill )
      Coil( #Warning.MaterialNotStandstill )
   END_RUNG
   // the same network as SCL:
   #Warning.MaterialNotStandstill := #COut.CutHead.Work_CheckNext AND #COut.DrawHead.Work_CheckNext AND #COut.MarkHead.Work_CheckNext AND NOT #CIn.MaterialStandstill;
END_REGION

REGION Network 54: >
END_REGION

REGION Network 55: >
END_REGION

REGION Network 56: <<<< FINAL >>>>
END_REGION

REGION Network 57: Coordination Out
   RUNG wire#powerrail
      { S7_Templates := "[card := 3, value_type := DInt]" } MAX(in1 := #HMI.CutHead.Avg_R_to_W_Time, in2 := #HMI.DrawHead.Avg_R_to_W_Time, in3 := #HMI.MarkHead.Avg_R_to_W_Time, out => #COut.Avg_R_to_W_Time)
   END_RUNG
   RUNG wire#powerrail
      { S7_Templates := "[card := 3, value_type := DInt]" } MAX(in1 := #HMI.CutHead.Avg_W_to_R_Time, in2 := #HMI.DrawHead.Avg_W_to_R_Time, in3 := #HMI.MarkHead.Avg_W_to_R_Time, out => #COut.Avg_W_to_R_Time)
   END_RUNG
   RUNG wire#powerrail
      Contact( #CutHead.COut.Rest )
      Contact( #DrawHead.COut.Rest )
      Contact( #MarkHead.COut.Rest )
      Contact( #Locking.COut.Work )
      Coil( #COut.AllAtRest )
   END_RUNG
   // the same network as SCL:
   #COut.Avg_R_to_W_Time := MAX(IN1 := #HMI.CutHead.Avg_R_to_W_Time, IN2 := #HMI.DrawHead.Avg_R_to_W_Time, IN3 := #HMI.MarkHead.Avg_R_to_W_Time);
   #COut.Avg_W_to_R_Time := MAX(IN1 := #HMI.CutHead.Avg_W_to_R_Time, IN2 := #HMI.DrawHead.Avg_W_to_R_Time, IN3 := #HMI.MarkHead.Avg_W_to_R_Time);
   #COut.AllAtRest := #CutHead.COut.Rest AND #DrawHead.COut.Rest AND #MarkHead.COut.Rest AND #Locking.COut.Work;
END_REGION

REGION Network 58: Collect machine to zone interface (internal machines OR)
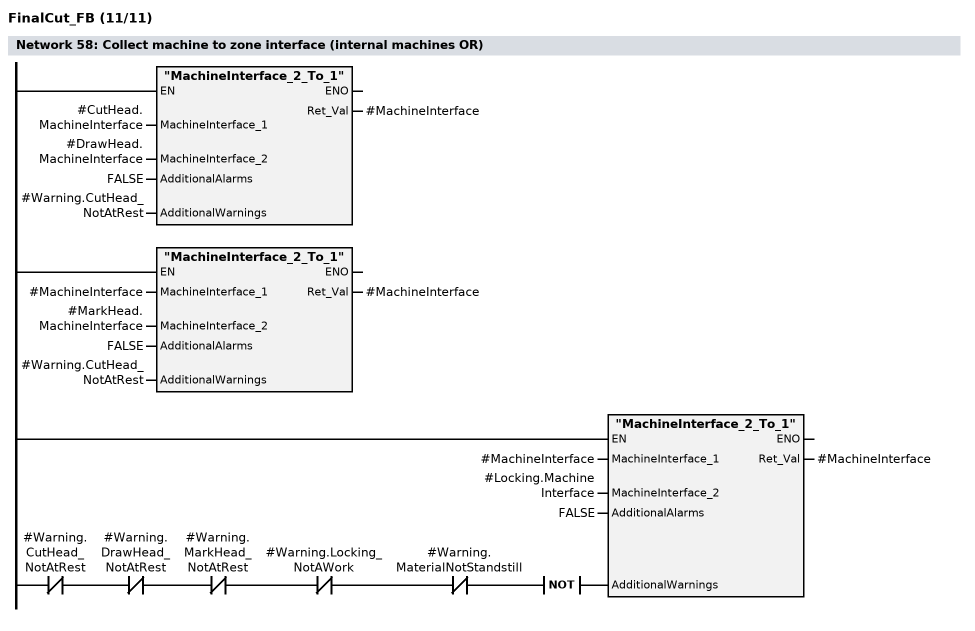
   RUNG wire#powerrail
      "MachineInterface_2_To_1"(MachineInterface_1 := #CutHead.MachineInterface, MachineInterface_2 := #DrawHead.MachineInterface, AdditionalAlarms := FALSE, AdditionalWarnings := #Warning.CutHead_NotAtRest, Ret_Val => #MachineInterface)
   END_RUNG
   RUNG wire#powerrail
      "MachineInterface_2_To_1"(MachineInterface_1 := #MachineInterface, MachineInterface_2 := #MarkHead.MachineInterface, AdditionalAlarms := FALSE, AdditionalWarnings := #Warning.CutHead_NotAtRest, Ret_Val => #MachineInterface)
   END_RUNG
   RUNG wire#powerrail
      "MachineInterface_2_To_1"(AdditionalWarnings := wire#w1, MachineInterface_1 := #MachineInterface, MachineInterface_2 := #Locking.MachineInterface, AdditionalAlarms := FALSE, Ret_Val => #MachineInterface)
   END_RUNG
   RUNG wire#powerrail
      I_Contact( #Warning.CutHead_NotAtRest )
      I_Contact( #Warning.DrawHead_NotAtRest )
      I_Contact( #Warning.MarkHead_NotAtRest )
      I_Contact( #Warning.Locking_NotAWork )
      I_Contact( #Warning.MaterialNotStandstill )
      Not()
   END_RUNG wire#w1
   // the same network as SCL:
   #MachineInterface := "MachineInterface_2_To_1"(MachineInterface_1 := #CutHead.MachineInterface,
                           MachineInterface_2 := #DrawHead.MachineInterface,
                           AdditionalAlarms := FALSE,
                           AdditionalWarnings := #Warning.CutHead_NotAtRest);
   #MachineInterface := "MachineInterface_2_To_1"(MachineInterface_1 := #MachineInterface,
                           MachineInterface_2 := #MarkHead.MachineInterface,
                           AdditionalAlarms := FALSE,
                           AdditionalWarnings := #Warning.CutHead_NotAtRest);
   #MachineInterface := "MachineInterface_2_To_1"(MachineInterface_1 := #MachineInterface,
                           MachineInterface_2 := #Locking.MachineInterface,
                           AdditionalAlarms := FALSE,
                           AdditionalWarnings := NOT (NOT #Warning.CutHead_NotAtRest AND NOT #Warning.DrawHead_NotAtRest AND NOT #Warning.MarkHead_NotAtRest AND NOT #Warning.Locking_NotAWork AND NOT #Warning.MaterialNotStandstill));
END_REGION
END_FUNCTION_BLOCK
